   // GBK_TO_UNICODE[17068] := 16#B57B;
   // GBK_TO_UNICODE[17069] := 16#7958;
   // GBK_TO_UNICODE[17070] := 16#B57C;
   // GBK_TO_UNICODE[17071] := 16#7959;
   // GBK_TO_UNICODE[17072] := 16#B57D;
   // GBK_TO_UNICODE[17073] := 16#7961;
   // GBK_TO_UNICODE[17074] := 16#B57E;
   // GBK_TO_UNICODE[17075] := 16#7963;
   // GBK_TO_UNICODE[17076] := 16#B580;
   // GBK_TO_UNICODE[17077] := 16#7964;
   // GBK_TO_UNICODE[17078] := 16#B581;
   // GBK_TO_UNICODE[17079] := 16#7966;
   // GBK_TO_UNICODE[17080] := 16#B582;
   // GBK_TO_UNICODE[17081] := 16#7969;
   // GBK_TO_UNICODE[17082] := 16#B583;
   // GBK_TO_UNICODE[17083] := 16#796A;
   // GBK_TO_UNICODE[17084] := 16#B584;
   // GBK_TO_UNICODE[17085] := 16#796B;
   // GBK_TO_UNICODE[17086] := 16#B585;
   // GBK_TO_UNICODE[17087] := 16#796C;
   // GBK_TO_UNICODE[17088] := 16#B586;
   // GBK_TO_UNICODE[17089] := 16#796E;
   // GBK_TO_UNICODE[17090] := 16#B587;
   // GBK_TO_UNICODE[17091] := 16#7970;
   // GBK_TO_UNICODE[17092] := 16#B588;
   // GBK_TO_UNICODE[17093] := 16#7971;
   // GBK_TO_UNICODE[17094] := 16#B589;
   // GBK_TO_UNICODE[17095] := 16#7972;
   // GBK_TO_UNICODE[17096] := 16#B58A;
   // GBK_TO_UNICODE[17097] := 16#7973;
   // GBK_TO_UNICODE[17098] := 16#B58B;
   // GBK_TO_UNICODE[17099] := 16#7974;
   // GBK_TO_UNICODE[17100] := 16#B58C;
   // GBK_TO_UNICODE[17101] := 16#7975;
   // GBK_TO_UNICODE[17102] := 16#B58D;
   // GBK_TO_UNICODE[17103] := 16#7976;
   // GBK_TO_UNICODE[17104] := 16#B58E;
   // GBK_TO_UNICODE[17105] := 16#7979;
   // GBK_TO_UNICODE[17106] := 16#B58F;
   // GBK_TO_UNICODE[17107] := 16#797B;
   // GBK_TO_UNICODE[17108] := 16#B590;
   // GBK_TO_UNICODE[17109] := 16#797C;
   // GBK_TO_UNICODE[17110] := 16#B591;
   // GBK_TO_UNICODE[17111] := 16#797D;
   // GBK_TO_UNICODE[17112] := 16#B592;
   // GBK_TO_UNICODE[17113] := 16#797E;
   // GBK_TO_UNICODE[17114] := 16#B593;
   // GBK_TO_UNICODE[17115] := 16#797F;
   // GBK_TO_UNICODE[17116] := 16#B594;
   // GBK_TO_UNICODE[17117] := 16#7982;
   // GBK_TO_UNICODE[17118] := 16#B595;
   // GBK_TO_UNICODE[17119] := 16#7983;
   // GBK_TO_UNICODE[17120] := 16#B596;
   // GBK_TO_UNICODE[17121] := 16#7986;
   // GBK_TO_UNICODE[17122] := 16#B597;
   // GBK_TO_UNICODE[17123] := 16#7987;
   // GBK_TO_UNICODE[17124] := 16#B598;
   // GBK_TO_UNICODE[17125] := 16#7988;
   // GBK_TO_UNICODE[17126] := 16#B599;
   // GBK_TO_UNICODE[17127] := 16#7989;
   // GBK_TO_UNICODE[17128] := 16#B59A;
   // GBK_TO_UNICODE[17129] := 16#798B;
   // GBK_TO_UNICODE[17130] := 16#B59B;
   // GBK_TO_UNICODE[17131] := 16#798C;
   // GBK_TO_UNICODE[17132] := 16#B59C;
   // GBK_TO_UNICODE[17133] := 16#798D;
   // GBK_TO_UNICODE[17134] := 16#B59D;
   // GBK_TO_UNICODE[17135] := 16#798E;
   // GBK_TO_UNICODE[17136] := 16#B59E;
   // GBK_TO_UNICODE[17137] := 16#7990;
   // GBK_TO_UNICODE[17138] := 16#B59F;
   // GBK_TO_UNICODE[17139] := 16#7991;
   // GBK_TO_UNICODE[17140] := 16#B5A0;
   // GBK_TO_UNICODE[17141] := 16#7992;
   // GBK_TO_UNICODE[17142] := 16#B5A1;
   // GBK_TO_UNICODE[17143] := 16#6020;
   // GBK_TO_UNICODE[17144] := 16#B5A2;
   // GBK_TO_UNICODE[17145] := 16#803D;
   // GBK_TO_UNICODE[17146] := 16#B5A3;
   // GBK_TO_UNICODE[17147] := 16#62C5;
   // GBK_TO_UNICODE[17148] := 16#B5A4;
   // GBK_TO_UNICODE[17149] := 16#4E39;
   // GBK_TO_UNICODE[17150] := 16#B5A5;
   // GBK_TO_UNICODE[17151] := 16#5355;
   // GBK_TO_UNICODE[17152] := 16#B5A6;
   // GBK_TO_UNICODE[17153] := 16#90F8;
   // GBK_TO_UNICODE[17154] := 16#B5A7;
   // GBK_TO_UNICODE[17155] := 16#63B8;
   // GBK_TO_UNICODE[17156] := 16#B5A8;
   // GBK_TO_UNICODE[17157] := 16#80C6;
   // GBK_TO_UNICODE[17158] := 16#B5A9;
   // GBK_TO_UNICODE[17159] := 16#65E6;
   // GBK_TO_UNICODE[17160] := 16#B5AA;
   // GBK_TO_UNICODE[17161] := 16#6C2E;
   // GBK_TO_UNICODE[17162] := 16#B5AB;
   // GBK_TO_UNICODE[17163] := 16#4F46;
   // GBK_TO_UNICODE[17164] := 16#B5AC;
   // GBK_TO_UNICODE[17165] := 16#60EE;
   // GBK_TO_UNICODE[17166] := 16#B5AD;
   // GBK_TO_UNICODE[17167] := 16#6DE1;
   // GBK_TO_UNICODE[17168] := 16#B5AE;
   // GBK_TO_UNICODE[17169] := 16#8BDE;
   // GBK_TO_UNICODE[17170] := 16#B5AF;
   // GBK_TO_UNICODE[17171] := 16#5F39;
   // GBK_TO_UNICODE[17172] := 16#B5B0;
   // GBK_TO_UNICODE[17173] := 16#86CB;
   // GBK_TO_UNICODE[17174] := 16#B5B1;
   // GBK_TO_UNICODE[17175] := 16#5F53;
   // GBK_TO_UNICODE[17176] := 16#B5B2;
   // GBK_TO_UNICODE[17177] := 16#6321;
   // GBK_TO_UNICODE[17178] := 16#B5B3;
   // GBK_TO_UNICODE[17179] := 16#515A;
   // GBK_TO_UNICODE[17180] := 16#B5B4;
   // GBK_TO_UNICODE[17181] := 16#8361;
   // GBK_TO_UNICODE[17182] := 16#B5B5;
   // GBK_TO_UNICODE[17183] := 16#6863;
   // GBK_TO_UNICODE[17184] := 16#B5B6;
   // GBK_TO_UNICODE[17185] := 16#5200;
   // GBK_TO_UNICODE[17186] := 16#B5B7;
   // GBK_TO_UNICODE[17187] := 16#6363;
   // GBK_TO_UNICODE[17188] := 16#B5B8;
   // GBK_TO_UNICODE[17189] := 16#8E48;
   // GBK_TO_UNICODE[17190] := 16#B5B9;
   // GBK_TO_UNICODE[17191] := 16#5012;
   // GBK_TO_UNICODE[17192] := 16#B5BA;
   // GBK_TO_UNICODE[17193] := 16#5C9B;
   // GBK_TO_UNICODE[17194] := 16#B5BB;
   // GBK_TO_UNICODE[17195] := 16#7977;
   // GBK_TO_UNICODE[17196] := 16#B5BC;
   // GBK_TO_UNICODE[17197] := 16#5BFC;
   // GBK_TO_UNICODE[17198] := 16#B5BD;
   // GBK_TO_UNICODE[17199] := 16#5230;
   // GBK_TO_UNICODE[17200] := 16#B5BE;
   // GBK_TO_UNICODE[17201] := 16#7A3B;
   // GBK_TO_UNICODE[17202] := 16#B5BF;
   // GBK_TO_UNICODE[17203] := 16#60BC;
   // GBK_TO_UNICODE[17204] := 16#B5C0;
   // GBK_TO_UNICODE[17205] := 16#9053;
   // GBK_TO_UNICODE[17206] := 16#B5C1;
   // GBK_TO_UNICODE[17207] := 16#76D7;
   // GBK_TO_UNICODE[17208] := 16#B5C2;
   // GBK_TO_UNICODE[17209] := 16#5FB7;
   // GBK_TO_UNICODE[17210] := 16#B5C3;
   // GBK_TO_UNICODE[17211] := 16#5F97;
   // GBK_TO_UNICODE[17212] := 16#B5C4;
   // GBK_TO_UNICODE[17213] := 16#7684;
   // GBK_TO_UNICODE[17214] := 16#B5C5;
   // GBK_TO_UNICODE[17215] := 16#8E6C;
   // GBK_TO_UNICODE[17216] := 16#B5C6;
   // GBK_TO_UNICODE[17217] := 16#706F;
   // GBK_TO_UNICODE[17218] := 16#B5C7;
   // GBK_TO_UNICODE[17219] := 16#767B;
   // GBK_TO_UNICODE[17220] := 16#B5C8;
   // GBK_TO_UNICODE[17221] := 16#7B49;
   // GBK_TO_UNICODE[17222] := 16#B5C9;
   // GBK_TO_UNICODE[17223] := 16#77AA;
   // GBK_TO_UNICODE[17224] := 16#B5CA;
   // GBK_TO_UNICODE[17225] := 16#51F3;
   // GBK_TO_UNICODE[17226] := 16#B5CB;
   // GBK_TO_UNICODE[17227] := 16#9093;
   // GBK_TO_UNICODE[17228] := 16#B5CC;
   // GBK_TO_UNICODE[17229] := 16#5824;
   // GBK_TO_UNICODE[17230] := 16#B5CD;
   // GBK_TO_UNICODE[17231] := 16#4F4E;
   // GBK_TO_UNICODE[17232] := 16#B5CE;
   // GBK_TO_UNICODE[17233] := 16#6EF4;
   // GBK_TO_UNICODE[17234] := 16#B5CF;
   // GBK_TO_UNICODE[17235] := 16#8FEA;
   // GBK_TO_UNICODE[17236] := 16#B5D0;
   // GBK_TO_UNICODE[17237] := 16#654C;
   // GBK_TO_UNICODE[17238] := 16#B5D1;
   // GBK_TO_UNICODE[17239] := 16#7B1B;
   // GBK_TO_UNICODE[17240] := 16#B5D2;
   // GBK_TO_UNICODE[17241] := 16#72C4;
   // GBK_TO_UNICODE[17242] := 16#B5D3;
   // GBK_TO_UNICODE[17243] := 16#6DA4;
   // GBK_TO_UNICODE[17244] := 16#B5D4;
   // GBK_TO_UNICODE[17245] := 16#7FDF;
   // GBK_TO_UNICODE[17246] := 16#B5D5;
   // GBK_TO_UNICODE[17247] := 16#5AE1;
   // GBK_TO_UNICODE[17248] := 16#B5D6;
   // GBK_TO_UNICODE[17249] := 16#62B5;
   // GBK_TO_UNICODE[17250] := 16#B5D7;
   // GBK_TO_UNICODE[17251] := 16#5E95;
   // GBK_TO_UNICODE[17252] := 16#B5D8;
   // GBK_TO_UNICODE[17253] := 16#5730;
   // GBK_TO_UNICODE[17254] := 16#B5D9;
   // GBK_TO_UNICODE[17255] := 16#8482;
   // GBK_TO_UNICODE[17256] := 16#B5DA;
   // GBK_TO_UNICODE[17257] := 16#7B2C;
   // GBK_TO_UNICODE[17258] := 16#B5DB;
   // GBK_TO_UNICODE[17259] := 16#5E1D;
   // GBK_TO_UNICODE[17260] := 16#B5DC;
   // GBK_TO_UNICODE[17261] := 16#5F1F;
   // GBK_TO_UNICODE[17262] := 16#B5DD;
   // GBK_TO_UNICODE[17263] := 16#9012;
   // GBK_TO_UNICODE[17264] := 16#B5DE;
   // GBK_TO_UNICODE[17265] := 16#7F14;
   // GBK_TO_UNICODE[17266] := 16#B5DF;
   // GBK_TO_UNICODE[17267] := 16#98A0;
   // GBK_TO_UNICODE[17268] := 16#B5E0;
   // GBK_TO_UNICODE[17269] := 16#6382;
   // GBK_TO_UNICODE[17270] := 16#B5E1;
   // GBK_TO_UNICODE[17271] := 16#6EC7;
   // GBK_TO_UNICODE[17272] := 16#B5E2;
   // GBK_TO_UNICODE[17273] := 16#7898;
   // GBK_TO_UNICODE[17274] := 16#B5E3;
   // GBK_TO_UNICODE[17275] := 16#70B9;
   // GBK_TO_UNICODE[17276] := 16#B5E4;
   // GBK_TO_UNICODE[17277] := 16#5178;
   // GBK_TO_UNICODE[17278] := 16#B5E5;
   // GBK_TO_UNICODE[17279] := 16#975B;
   // GBK_TO_UNICODE[17280] := 16#B5E6;
   // GBK_TO_UNICODE[17281] := 16#57AB;
   // GBK_TO_UNICODE[17282] := 16#B5E7;
   // GBK_TO_UNICODE[17283] := 16#7535;
   // GBK_TO_UNICODE[17284] := 16#B5E8;
   // GBK_TO_UNICODE[17285] := 16#4F43;
   // GBK_TO_UNICODE[17286] := 16#B5E9;
   // GBK_TO_UNICODE[17287] := 16#7538;
   // GBK_TO_UNICODE[17288] := 16#B5EA;
   // GBK_TO_UNICODE[17289] := 16#5E97;
   // GBK_TO_UNICODE[17290] := 16#B5EB;
   // GBK_TO_UNICODE[17291] := 16#60E6;
   // GBK_TO_UNICODE[17292] := 16#B5EC;
   // GBK_TO_UNICODE[17293] := 16#5960;
   // GBK_TO_UNICODE[17294] := 16#B5ED;
   // GBK_TO_UNICODE[17295] := 16#6DC0;
   // GBK_TO_UNICODE[17296] := 16#B5EE;
   // GBK_TO_UNICODE[17297] := 16#6BBF;
   // GBK_TO_UNICODE[17298] := 16#B5EF;
   // GBK_TO_UNICODE[17299] := 16#7889;
   // GBK_TO_UNICODE[17300] := 16#B5F0;
   // GBK_TO_UNICODE[17301] := 16#53FC;
   // GBK_TO_UNICODE[17302] := 16#B5F1;
   // GBK_TO_UNICODE[17303] := 16#96D5;
   // GBK_TO_UNICODE[17304] := 16#B5F2;
   // GBK_TO_UNICODE[17305] := 16#51CB;
   // GBK_TO_UNICODE[17306] := 16#B5F3;
   // GBK_TO_UNICODE[17307] := 16#5201;
   // GBK_TO_UNICODE[17308] := 16#B5F4;
   // GBK_TO_UNICODE[17309] := 16#6389;
   // GBK_TO_UNICODE[17310] := 16#B5F5;
   // GBK_TO_UNICODE[17311] := 16#540A;
   // GBK_TO_UNICODE[17312] := 16#B5F6;
   // GBK_TO_UNICODE[17313] := 16#9493;
   // GBK_TO_UNICODE[17314] := 16#B5F7;
   // GBK_TO_UNICODE[17315] := 16#8C03;
   // GBK_TO_UNICODE[17316] := 16#B5F8;
   // GBK_TO_UNICODE[17317] := 16#8DCC;
   // GBK_TO_UNICODE[17318] := 16#B5F9;
   // GBK_TO_UNICODE[17319] := 16#7239;
   // GBK_TO_UNICODE[17320] := 16#B5FA;
   // GBK_TO_UNICODE[17321] := 16#789F;
   // GBK_TO_UNICODE[17322] := 16#B5FB;
   // GBK_TO_UNICODE[17323] := 16#8776;
   // GBK_TO_UNICODE[17324] := 16#B5FC;
   // GBK_TO_UNICODE[17325] := 16#8FED;
   // GBK_TO_UNICODE[17326] := 16#B5FD;
   // GBK_TO_UNICODE[17327] := 16#8C0D;
   // GBK_TO_UNICODE[17328] := 16#B5FE;
   // GBK_TO_UNICODE[17329] := 16#53E0;
   // GBK_TO_UNICODE[17330] := 16#B640;
   // GBK_TO_UNICODE[17331] := 16#7993;
   // GBK_TO_UNICODE[17332] := 16#B641;
   // GBK_TO_UNICODE[17333] := 16#7994;
   // GBK_TO_UNICODE[17334] := 16#B642;
   // GBK_TO_UNICODE[17335] := 16#7995;
   // GBK_TO_UNICODE[17336] := 16#B643;
   // GBK_TO_UNICODE[17337] := 16#7996;
   // GBK_TO_UNICODE[17338] := 16#B644;
   // GBK_TO_UNICODE[17339] := 16#7997;
   // GBK_TO_UNICODE[17340] := 16#B645;
   // GBK_TO_UNICODE[17341] := 16#7998;
   // GBK_TO_UNICODE[17342] := 16#B646;
   // GBK_TO_UNICODE[17343] := 16#7999;
   // GBK_TO_UNICODE[17344] := 16#B647;
   // GBK_TO_UNICODE[17345] := 16#799B;
   // GBK_TO_UNICODE[17346] := 16#B648;
   // GBK_TO_UNICODE[17347] := 16#799C;
   // GBK_TO_UNICODE[17348] := 16#B649;
   // GBK_TO_UNICODE[17349] := 16#799D;
   // GBK_TO_UNICODE[17350] := 16#B64A;
   // GBK_TO_UNICODE[17351] := 16#799E;
   // GBK_TO_UNICODE[17352] := 16#B64B;
   // GBK_TO_UNICODE[17353] := 16#799F;
   // GBK_TO_UNICODE[17354] := 16#B64C;
   // GBK_TO_UNICODE[17355] := 16#79A0;
   // GBK_TO_UNICODE[17356] := 16#B64D;
   // GBK_TO_UNICODE[17357] := 16#79A1;
   // GBK_TO_UNICODE[17358] := 16#B64E;
   // GBK_TO_UNICODE[17359] := 16#79A2;
   // GBK_TO_UNICODE[17360] := 16#B64F;
   // GBK_TO_UNICODE[17361] := 16#79A3;
   // GBK_TO_UNICODE[17362] := 16#B650;
   // GBK_TO_UNICODE[17363] := 16#79A4;
   // GBK_TO_UNICODE[17364] := 16#B651;
   // GBK_TO_UNICODE[17365] := 16#79A5;
   // GBK_TO_UNICODE[17366] := 16#B652;
   // GBK_TO_UNICODE[17367] := 16#79A6;
   // GBK_TO_UNICODE[17368] := 16#B653;
   // GBK_TO_UNICODE[17369] := 16#79A8;
   // GBK_TO_UNICODE[17370] := 16#B654;
   // GBK_TO_UNICODE[17371] := 16#79A9;
   // GBK_TO_UNICODE[17372] := 16#B655;
   // GBK_TO_UNICODE[17373] := 16#79AA;
   // GBK_TO_UNICODE[17374] := 16#B656;
   // GBK_TO_UNICODE[17375] := 16#79AB;
   // GBK_TO_UNICODE[17376] := 16#B657;
   // GBK_TO_UNICODE[17377] := 16#79AC;
   // GBK_TO_UNICODE[17378] := 16#B658;
   // GBK_TO_UNICODE[17379] := 16#79AD;
   // GBK_TO_UNICODE[17380] := 16#B659;
   // GBK_TO_UNICODE[17381] := 16#79AE;
   // GBK_TO_UNICODE[17382] := 16#B65A;
   // GBK_TO_UNICODE[17383] := 16#79AF;
   // GBK_TO_UNICODE[17384] := 16#B65B;
   // GBK_TO_UNICODE[17385] := 16#79B0;
   // GBK_TO_UNICODE[17386] := 16#B65C;
   // GBK_TO_UNICODE[17387] := 16#79B1;
   // GBK_TO_UNICODE[17388] := 16#B65D;
   // GBK_TO_UNICODE[17389] := 16#79B2;
   // GBK_TO_UNICODE[17390] := 16#B65E;
   // GBK_TO_UNICODE[17391] := 16#79B4;
   // GBK_TO_UNICODE[17392] := 16#B65F;
   // GBK_TO_UNICODE[17393] := 16#79B5;
   // GBK_TO_UNICODE[17394] := 16#B660;
   // GBK_TO_UNICODE[17395] := 16#79B6;
   // GBK_TO_UNICODE[17396] := 16#B661;
   // GBK_TO_UNICODE[17397] := 16#79B7;
   // GBK_TO_UNICODE[17398] := 16#B662;
   // GBK_TO_UNICODE[17399] := 16#79B8;
   // GBK_TO_UNICODE[17400] := 16#B663;
   // GBK_TO_UNICODE[17401] := 16#79BC;
   // GBK_TO_UNICODE[17402] := 16#B664;
   // GBK_TO_UNICODE[17403] := 16#79BF;
   // GBK_TO_UNICODE[17404] := 16#B665;
   // GBK_TO_UNICODE[17405] := 16#79C2;
   // GBK_TO_UNICODE[17406] := 16#B666;
   // GBK_TO_UNICODE[17407] := 16#79C4;
   // GBK_TO_UNICODE[17408] := 16#B667;
   // GBK_TO_UNICODE[17409] := 16#79C5;
   // GBK_TO_UNICODE[17410] := 16#B668;
   // GBK_TO_UNICODE[17411] := 16#79C7;
   // GBK_TO_UNICODE[17412] := 16#B669;
   // GBK_TO_UNICODE[17413] := 16#79C8;
   // GBK_TO_UNICODE[17414] := 16#B66A;
   // GBK_TO_UNICODE[17415] := 16#79CA;
   // GBK_TO_UNICODE[17416] := 16#B66B;
   // GBK_TO_UNICODE[17417] := 16#79CC;
   // GBK_TO_UNICODE[17418] := 16#B66C;
   // GBK_TO_UNICODE[17419] := 16#79CE;
   // GBK_TO_UNICODE[17420] := 16#B66D;
   // GBK_TO_UNICODE[17421] := 16#79CF;
   // GBK_TO_UNICODE[17422] := 16#B66E;
   // GBK_TO_UNICODE[17423] := 16#79D0;
   // GBK_TO_UNICODE[17424] := 16#B66F;
   // GBK_TO_UNICODE[17425] := 16#79D3;
   // GBK_TO_UNICODE[17426] := 16#B670;
   // GBK_TO_UNICODE[17427] := 16#79D4;
   // GBK_TO_UNICODE[17428] := 16#B671;
   // GBK_TO_UNICODE[17429] := 16#79D6;
   // GBK_TO_UNICODE[17430] := 16#B672;
   // GBK_TO_UNICODE[17431] := 16#79D7;
   // GBK_TO_UNICODE[17432] := 16#B673;
   // GBK_TO_UNICODE[17433] := 16#79D9;
   // GBK_TO_UNICODE[17434] := 16#B674;
   // GBK_TO_UNICODE[17435] := 16#79DA;
   // GBK_TO_UNICODE[17436] := 16#B675;
   // GBK_TO_UNICODE[17437] := 16#79DB;
   // GBK_TO_UNICODE[17438] := 16#B676;
   // GBK_TO_UNICODE[17439] := 16#79DC;
   // GBK_TO_UNICODE[17440] := 16#B677;
   // GBK_TO_UNICODE[17441] := 16#79DD;
   // GBK_TO_UNICODE[17442] := 16#B678;
   // GBK_TO_UNICODE[17443] := 16#79DE;
   // GBK_TO_UNICODE[17444] := 16#B679;
   // GBK_TO_UNICODE[17445] := 16#79E0;
   // GBK_TO_UNICODE[17446] := 16#B67A;
   // GBK_TO_UNICODE[17447] := 16#79E1;
   // GBK_TO_UNICODE[17448] := 16#B67B;
   // GBK_TO_UNICODE[17449] := 16#79E2;
   // GBK_TO_UNICODE[17450] := 16#B67C;
   // GBK_TO_UNICODE[17451] := 16#79E5;
   // GBK_TO_UNICODE[17452] := 16#B67D;
   // GBK_TO_UNICODE[17453] := 16#79E8;
   // GBK_TO_UNICODE[17454] := 16#B67E;
   // GBK_TO_UNICODE[17455] := 16#79EA;
   // GBK_TO_UNICODE[17456] := 16#B680;
   // GBK_TO_UNICODE[17457] := 16#79EC;
   // GBK_TO_UNICODE[17458] := 16#B681;
   // GBK_TO_UNICODE[17459] := 16#79EE;
   // GBK_TO_UNICODE[17460] := 16#B682;
   // GBK_TO_UNICODE[17461] := 16#79F1;
   // GBK_TO_UNICODE[17462] := 16#B683;
   // GBK_TO_UNICODE[17463] := 16#79F2;
   // GBK_TO_UNICODE[17464] := 16#B684;
   // GBK_TO_UNICODE[17465] := 16#79F3;
   // GBK_TO_UNICODE[17466] := 16#B685;
   // GBK_TO_UNICODE[17467] := 16#79F4;
   // GBK_TO_UNICODE[17468] := 16#B686;
   // GBK_TO_UNICODE[17469] := 16#79F5;
   // GBK_TO_UNICODE[17470] := 16#B687;
   // GBK_TO_UNICODE[17471] := 16#79F6;
   // GBK_TO_UNICODE[17472] := 16#B688;
   // GBK_TO_UNICODE[17473] := 16#79F7;
   // GBK_TO_UNICODE[17474] := 16#B689;
   // GBK_TO_UNICODE[17475] := 16#79F9;
   // GBK_TO_UNICODE[17476] := 16#B68A;
   // GBK_TO_UNICODE[17477] := 16#79FA;
   // GBK_TO_UNICODE[17478] := 16#B68B;
   // GBK_TO_UNICODE[17479] := 16#79FC;
   // GBK_TO_UNICODE[17480] := 16#B68C;
   // GBK_TO_UNICODE[17481] := 16#79FE;
   // GBK_TO_UNICODE[17482] := 16#B68D;
   // GBK_TO_UNICODE[17483] := 16#79FF;
   // GBK_TO_UNICODE[17484] := 16#B68E;
   // GBK_TO_UNICODE[17485] := 16#7A01;
   // GBK_TO_UNICODE[17486] := 16#B68F;
   // GBK_TO_UNICODE[17487] := 16#7A04;
   // GBK_TO_UNICODE[17488] := 16#B690;
   // GBK_TO_UNICODE[17489] := 16#7A05;
   // GBK_TO_UNICODE[17490] := 16#B691;
   // GBK_TO_UNICODE[17491] := 16#7A07;
   // GBK_TO_UNICODE[17492] := 16#B692;
   // GBK_TO_UNICODE[17493] := 16#7A08;
   // GBK_TO_UNICODE[17494] := 16#B693;
   // GBK_TO_UNICODE[17495] := 16#7A09;
   // GBK_TO_UNICODE[17496] := 16#B694;
   // GBK_TO_UNICODE[17497] := 16#7A0A;
   // GBK_TO_UNICODE[17498] := 16#B695;
   // GBK_TO_UNICODE[17499] := 16#7A0C;
   // GBK_TO_UNICODE[17500] := 16#B696;
   // GBK_TO_UNICODE[17501] := 16#7A0F;
   // GBK_TO_UNICODE[17502] := 16#B697;
   // GBK_TO_UNICODE[17503] := 16#7A10;
   // GBK_TO_UNICODE[17504] := 16#B698;
   // GBK_TO_UNICODE[17505] := 16#7A11;
   // GBK_TO_UNICODE[17506] := 16#B699;
   // GBK_TO_UNICODE[17507] := 16#7A12;
   // GBK_TO_UNICODE[17508] := 16#B69A;
   // GBK_TO_UNICODE[17509] := 16#7A13;
   // GBK_TO_UNICODE[17510] := 16#B69B;
   // GBK_TO_UNICODE[17511] := 16#7A15;
   // GBK_TO_UNICODE[17512] := 16#B69C;
   // GBK_TO_UNICODE[17513] := 16#7A16;
   // GBK_TO_UNICODE[17514] := 16#B69D;
   // GBK_TO_UNICODE[17515] := 16#7A18;
   // GBK_TO_UNICODE[17516] := 16#B69E;
   // GBK_TO_UNICODE[17517] := 16#7A19;
   // GBK_TO_UNICODE[17518] := 16#B69F;
   // GBK_TO_UNICODE[17519] := 16#7A1B;
   // GBK_TO_UNICODE[17520] := 16#B6A0;
   // GBK_TO_UNICODE[17521] := 16#7A1C;
   // GBK_TO_UNICODE[17522] := 16#B6A1;
   // GBK_TO_UNICODE[17523] := 16#4E01;
   // GBK_TO_UNICODE[17524] := 16#B6A2;
   // GBK_TO_UNICODE[17525] := 16#76EF;
   // GBK_TO_UNICODE[17526] := 16#B6A3;
   // GBK_TO_UNICODE[17527] := 16#53EE;
   // GBK_TO_UNICODE[17528] := 16#B6A4;
   // GBK_TO_UNICODE[17529] := 16#9489;
   // GBK_TO_UNICODE[17530] := 16#B6A5;
   // GBK_TO_UNICODE[17531] := 16#9876;
   // GBK_TO_UNICODE[17532] := 16#B6A6;
   // GBK_TO_UNICODE[17533] := 16#9F0E;
   // GBK_TO_UNICODE[17534] := 16#B6A7;
   // GBK_TO_UNICODE[17535] := 16#952D;
   // GBK_TO_UNICODE[17536] := 16#B6A8;
   // GBK_TO_UNICODE[17537] := 16#5B9A;
   // GBK_TO_UNICODE[17538] := 16#B6A9;
   // GBK_TO_UNICODE[17539] := 16#8BA2;
   // GBK_TO_UNICODE[17540] := 16#B6AA;
   // GBK_TO_UNICODE[17541] := 16#4E22;
   // GBK_TO_UNICODE[17542] := 16#B6AB;
   // GBK_TO_UNICODE[17543] := 16#4E1C;
   // GBK_TO_UNICODE[17544] := 16#B6AC;
   // GBK_TO_UNICODE[17545] := 16#51AC;
   // GBK_TO_UNICODE[17546] := 16#B6AD;
   // GBK_TO_UNICODE[17547] := 16#8463;
   // GBK_TO_UNICODE[17548] := 16#B6AE;
   // GBK_TO_UNICODE[17549] := 16#61C2;
   // GBK_TO_UNICODE[17550] := 16#B6AF;
   // GBK_TO_UNICODE[17551] := 16#52A8;
   // GBK_TO_UNICODE[17552] := 16#B6B0;
   // GBK_TO_UNICODE[17553] := 16#680B;
   // GBK_TO_UNICODE[17554] := 16#B6B1;
   // GBK_TO_UNICODE[17555] := 16#4F97;
   // GBK_TO_UNICODE[17556] := 16#B6B2;
   // GBK_TO_UNICODE[17557] := 16#606B;
   // GBK_TO_UNICODE[17558] := 16#B6B3;
   // GBK_TO_UNICODE[17559] := 16#51BB;
   // GBK_TO_UNICODE[17560] := 16#B6B4;
   // GBK_TO_UNICODE[17561] := 16#6D1E;
   // GBK_TO_UNICODE[17562] := 16#B6B5;
   // GBK_TO_UNICODE[17563] := 16#515C;
   // GBK_TO_UNICODE[17564] := 16#B6B6;
   // GBK_TO_UNICODE[17565] := 16#6296;
   // GBK_TO_UNICODE[17566] := 16#B6B7;
   // GBK_TO_UNICODE[17567] := 16#6597;
   // GBK_TO_UNICODE[17568] := 16#B6B8;
   // GBK_TO_UNICODE[17569] := 16#9661;
   // GBK_TO_UNICODE[17570] := 16#B6B9;
   // GBK_TO_UNICODE[17571] := 16#8C46;
   // GBK_TO_UNICODE[17572] := 16#B6BA;
   // GBK_TO_UNICODE[17573] := 16#9017;
   // GBK_TO_UNICODE[17574] := 16#B6BB;
   // GBK_TO_UNICODE[17575] := 16#75D8;
   // GBK_TO_UNICODE[17576] := 16#B6BC;
   // GBK_TO_UNICODE[17577] := 16#90FD;
   // GBK_TO_UNICODE[17578] := 16#B6BD;
   // GBK_TO_UNICODE[17579] := 16#7763;
   // GBK_TO_UNICODE[17580] := 16#B6BE;
   // GBK_TO_UNICODE[17581] := 16#6BD2;
   // GBK_TO_UNICODE[17582] := 16#B6BF;
   // GBK_TO_UNICODE[17583] := 16#728A;
   // GBK_TO_UNICODE[17584] := 16#B6C0;
   // GBK_TO_UNICODE[17585] := 16#72EC;
   // GBK_TO_UNICODE[17586] := 16#B6C1;
   // GBK_TO_UNICODE[17587] := 16#8BFB;
   // GBK_TO_UNICODE[17588] := 16#B6C2;
   // GBK_TO_UNICODE[17589] := 16#5835;
   // GBK_TO_UNICODE[17590] := 16#B6C3;
   // GBK_TO_UNICODE[17591] := 16#7779;
   // GBK_TO_UNICODE[17592] := 16#B6C4;
   // GBK_TO_UNICODE[17593] := 16#8D4C;
   // GBK_TO_UNICODE[17594] := 16#B6C5;
   // GBK_TO_UNICODE[17595] := 16#675C;
   // GBK_TO_UNICODE[17596] := 16#B6C6;
   // GBK_TO_UNICODE[17597] := 16#9540;
   // GBK_TO_UNICODE[17598] := 16#B6C7;
   // GBK_TO_UNICODE[17599] := 16#809A;
   // GBK_TO_UNICODE[17600] := 16#B6C8;
   // GBK_TO_UNICODE[17601] := 16#5EA6;
   // GBK_TO_UNICODE[17602] := 16#B6C9;
   // GBK_TO_UNICODE[17603] := 16#6E21;
   // GBK_TO_UNICODE[17604] := 16#B6CA;
   // GBK_TO_UNICODE[17605] := 16#5992;
   // GBK_TO_UNICODE[17606] := 16#B6CB;
   // GBK_TO_UNICODE[17607] := 16#7AEF;
   // GBK_TO_UNICODE[17608] := 16#B6CC;
   // GBK_TO_UNICODE[17609] := 16#77ED;
   // GBK_TO_UNICODE[17610] := 16#B6CD;
   // GBK_TO_UNICODE[17611] := 16#953B;
   // GBK_TO_UNICODE[17612] := 16#B6CE;
   // GBK_TO_UNICODE[17613] := 16#6BB5;
   // GBK_TO_UNICODE[17614] := 16#B6CF;
   // GBK_TO_UNICODE[17615] := 16#65AD;
   // GBK_TO_UNICODE[17616] := 16#B6D0;
   // GBK_TO_UNICODE[17617] := 16#7F0E;
   // GBK_TO_UNICODE[17618] := 16#B6D1;
   // GBK_TO_UNICODE[17619] := 16#5806;
   // GBK_TO_UNICODE[17620] := 16#B6D2;
   // GBK_TO_UNICODE[17621] := 16#5151;
   // GBK_TO_UNICODE[17622] := 16#B6D3;
   // GBK_TO_UNICODE[17623] := 16#961F;
   // GBK_TO_UNICODE[17624] := 16#B6D4;
   // GBK_TO_UNICODE[17625] := 16#5BF9;
   // GBK_TO_UNICODE[17626] := 16#B6D5;
   // GBK_TO_UNICODE[17627] := 16#58A9;
   // GBK_TO_UNICODE[17628] := 16#B6D6;
   // GBK_TO_UNICODE[17629] := 16#5428;
   // GBK_TO_UNICODE[17630] := 16#B6D7;
   // GBK_TO_UNICODE[17631] := 16#8E72;
   // GBK_TO_UNICODE[17632] := 16#B6D8;
   // GBK_TO_UNICODE[17633] := 16#6566;
   // GBK_TO_UNICODE[17634] := 16#B6D9;
   // GBK_TO_UNICODE[17635] := 16#987F;
   // GBK_TO_UNICODE[17636] := 16#B6DA;
   // GBK_TO_UNICODE[17637] := 16#56E4;
   // GBK_TO_UNICODE[17638] := 16#B6DB;
   // GBK_TO_UNICODE[17639] := 16#949D;
   // GBK_TO_UNICODE[17640] := 16#B6DC;
   // GBK_TO_UNICODE[17641] := 16#76FE;
   // GBK_TO_UNICODE[17642] := 16#B6DD;
   // GBK_TO_UNICODE[17643] := 16#9041;
   // GBK_TO_UNICODE[17644] := 16#B6DE;
   // GBK_TO_UNICODE[17645] := 16#6387;
   // GBK_TO_UNICODE[17646] := 16#B6DF;
   // GBK_TO_UNICODE[17647] := 16#54C6;
   // GBK_TO_UNICODE[17648] := 16#B6E0;
   // GBK_TO_UNICODE[17649] := 16#591A;
   // GBK_TO_UNICODE[17650] := 16#B6E1;
   // GBK_TO_UNICODE[17651] := 16#593A;
   // GBK_TO_UNICODE[17652] := 16#B6E2;
   // GBK_TO_UNICODE[17653] := 16#579B;
   // GBK_TO_UNICODE[17654] := 16#B6E3;
   // GBK_TO_UNICODE[17655] := 16#8EB2;
   // GBK_TO_UNICODE[17656] := 16#B6E4;
   // GBK_TO_UNICODE[17657] := 16#6735;
   // GBK_TO_UNICODE[17658] := 16#B6E5;
   // GBK_TO_UNICODE[17659] := 16#8DFA;
   // GBK_TO_UNICODE[17660] := 16#B6E6;
   // GBK_TO_UNICODE[17661] := 16#8235;
   // GBK_TO_UNICODE[17662] := 16#B6E7;
   // GBK_TO_UNICODE[17663] := 16#5241;
   // GBK_TO_UNICODE[17664] := 16#B6E8;
   // GBK_TO_UNICODE[17665] := 16#60F0;
   // GBK_TO_UNICODE[17666] := 16#B6E9;
   // GBK_TO_UNICODE[17667] := 16#5815;
   // GBK_TO_UNICODE[17668] := 16#B6EA;
   // GBK_TO_UNICODE[17669] := 16#86FE;
   // GBK_TO_UNICODE[17670] := 16#B6EB;
   // GBK_TO_UNICODE[17671] := 16#5CE8;
   // GBK_TO_UNICODE[17672] := 16#B6EC;
   // GBK_TO_UNICODE[17673] := 16#9E45;
   // GBK_TO_UNICODE[17674] := 16#B6ED;
   // GBK_TO_UNICODE[17675] := 16#4FC4;
   // GBK_TO_UNICODE[17676] := 16#B6EE;
   // GBK_TO_UNICODE[17677] := 16#989D;
   // GBK_TO_UNICODE[17678] := 16#B6EF;
   // GBK_TO_UNICODE[17679] := 16#8BB9;
   // GBK_TO_UNICODE[17680] := 16#B6F0;
   // GBK_TO_UNICODE[17681] := 16#5A25;
   // GBK_TO_UNICODE[17682] := 16#B6F1;
   // GBK_TO_UNICODE[17683] := 16#6076;
   // GBK_TO_UNICODE[17684] := 16#B6F2;
   // GBK_TO_UNICODE[17685] := 16#5384;
   // GBK_TO_UNICODE[17686] := 16#B6F3;
   // GBK_TO_UNICODE[17687] := 16#627C;
   // GBK_TO_UNICODE[17688] := 16#B6F4;
   // GBK_TO_UNICODE[17689] := 16#904F;
   // GBK_TO_UNICODE[17690] := 16#B6F5;
   // GBK_TO_UNICODE[17691] := 16#9102;
   // GBK_TO_UNICODE[17692] := 16#B6F6;
   // GBK_TO_UNICODE[17693] := 16#997F;
   // GBK_TO_UNICODE[17694] := 16#B6F7;
   // GBK_TO_UNICODE[17695] := 16#6069;
   // GBK_TO_UNICODE[17696] := 16#B6F8;
   // GBK_TO_UNICODE[17697] := 16#800C;
   // GBK_TO_UNICODE[17698] := 16#B6F9;
   // GBK_TO_UNICODE[17699] := 16#513F;
   // GBK_TO_UNICODE[17700] := 16#B6FA;
   // GBK_TO_UNICODE[17701] := 16#8033;
   // GBK_TO_UNICODE[17702] := 16#B6FB;
   // GBK_TO_UNICODE[17703] := 16#5C14;
   // GBK_TO_UNICODE[17704] := 16#B6FC;
   // GBK_TO_UNICODE[17705] := 16#9975;
   // GBK_TO_UNICODE[17706] := 16#B6FD;
   // GBK_TO_UNICODE[17707] := 16#6D31;
   // GBK_TO_UNICODE[17708] := 16#B6FE;
   // GBK_TO_UNICODE[17709] := 16#4E8C;
   // GBK_TO_UNICODE[17710] := 16#B740;
   // GBK_TO_UNICODE[17711] := 16#7A1D;
   // GBK_TO_UNICODE[17712] := 16#B741;
   // GBK_TO_UNICODE[17713] := 16#7A1F;
   // GBK_TO_UNICODE[17714] := 16#B742;
   // GBK_TO_UNICODE[17715] := 16#7A21;
   // GBK_TO_UNICODE[17716] := 16#B743;
   // GBK_TO_UNICODE[17717] := 16#7A22;
   // GBK_TO_UNICODE[17718] := 16#B744;
   // GBK_TO_UNICODE[17719] := 16#7A24;
   // GBK_TO_UNICODE[17720] := 16#B745;
   // GBK_TO_UNICODE[17721] := 16#7A25;
   // GBK_TO_UNICODE[17722] := 16#B746;
   // GBK_TO_UNICODE[17723] := 16#7A26;
   // GBK_TO_UNICODE[17724] := 16#B747;
   // GBK_TO_UNICODE[17725] := 16#7A27;
   // GBK_TO_UNICODE[17726] := 16#B748;
   // GBK_TO_UNICODE[17727] := 16#7A28;
   // GBK_TO_UNICODE[17728] := 16#B749;
   // GBK_TO_UNICODE[17729] := 16#7A29;
   // GBK_TO_UNICODE[17730] := 16#B74A;
   // GBK_TO_UNICODE[17731] := 16#7A2A;
   // GBK_TO_UNICODE[17732] := 16#B74B;
   // GBK_TO_UNICODE[17733] := 16#7A2B;
   // GBK_TO_UNICODE[17734] := 16#B74C;
   // GBK_TO_UNICODE[17735] := 16#7A2C;
   // GBK_TO_UNICODE[17736] := 16#B74D;
   // GBK_TO_UNICODE[17737] := 16#7A2D;
   // GBK_TO_UNICODE[17738] := 16#B74E;
   // GBK_TO_UNICODE[17739] := 16#7A2E;
   // GBK_TO_UNICODE[17740] := 16#B74F;
   // GBK_TO_UNICODE[17741] := 16#7A2F;
   // GBK_TO_UNICODE[17742] := 16#B750;
   // GBK_TO_UNICODE[17743] := 16#7A30;
   // GBK_TO_UNICODE[17744] := 16#B751;
   // GBK_TO_UNICODE[17745] := 16#7A31;
   // GBK_TO_UNICODE[17746] := 16#B752;
   // GBK_TO_UNICODE[17747] := 16#7A32;
   // GBK_TO_UNICODE[17748] := 16#B753;
   // GBK_TO_UNICODE[17749] := 16#7A34;
   // GBK_TO_UNICODE[17750] := 16#B754;
   // GBK_TO_UNICODE[17751] := 16#7A35;
   // GBK_TO_UNICODE[17752] := 16#B755;
   // GBK_TO_UNICODE[17753] := 16#7A36;
   // GBK_TO_UNICODE[17754] := 16#B756;
   // GBK_TO_UNICODE[17755] := 16#7A38;
   // GBK_TO_UNICODE[17756] := 16#B757;
   // GBK_TO_UNICODE[17757] := 16#7A3A;
   // GBK_TO_UNICODE[17758] := 16#B758;
   // GBK_TO_UNICODE[17759] := 16#7A3E;
   // GBK_TO_UNICODE[17760] := 16#B759;
   // GBK_TO_UNICODE[17761] := 16#7A40;
   // GBK_TO_UNICODE[17762] := 16#B75A;
   // GBK_TO_UNICODE[17763] := 16#7A41;
   // GBK_TO_UNICODE[17764] := 16#B75B;
   // GBK_TO_UNICODE[17765] := 16#7A42;
   // GBK_TO_UNICODE[17766] := 16#B75C;
   // GBK_TO_UNICODE[17767] := 16#7A43;
   // GBK_TO_UNICODE[17768] := 16#B75D;
   // GBK_TO_UNICODE[17769] := 16#7A44;
   // GBK_TO_UNICODE[17770] := 16#B75E;
   // GBK_TO_UNICODE[17771] := 16#7A45;
   // GBK_TO_UNICODE[17772] := 16#B75F;
   // GBK_TO_UNICODE[17773] := 16#7A47;
   // GBK_TO_UNICODE[17774] := 16#B760;
   // GBK_TO_UNICODE[17775] := 16#7A48;
   // GBK_TO_UNICODE[17776] := 16#B761;
   // GBK_TO_UNICODE[17777] := 16#7A49;
   // GBK_TO_UNICODE[17778] := 16#B762;
   // GBK_TO_UNICODE[17779] := 16#7A4A;
   // GBK_TO_UNICODE[17780] := 16#B763;
   // GBK_TO_UNICODE[17781] := 16#7A4B;
   // GBK_TO_UNICODE[17782] := 16#B764;
   // GBK_TO_UNICODE[17783] := 16#7A4C;
   // GBK_TO_UNICODE[17784] := 16#B765;
   // GBK_TO_UNICODE[17785] := 16#7A4D;
   // GBK_TO_UNICODE[17786] := 16#B766;
   // GBK_TO_UNICODE[17787] := 16#7A4E;
   // GBK_TO_UNICODE[17788] := 16#B767;
   // GBK_TO_UNICODE[17789] := 16#7A4F;
   // GBK_TO_UNICODE[17790] := 16#B768;
   // GBK_TO_UNICODE[17791] := 16#7A50;
   // GBK_TO_UNICODE[17792] := 16#B769;
   // GBK_TO_UNICODE[17793] := 16#7A52;
   // GBK_TO_UNICODE[17794] := 16#B76A;
   // GBK_TO_UNICODE[17795] := 16#7A53;
   // GBK_TO_UNICODE[17796] := 16#B76B;
   // GBK_TO_UNICODE[17797] := 16#7A54;
   // GBK_TO_UNICODE[17798] := 16#B76C;
   // GBK_TO_UNICODE[17799] := 16#7A55;
   // GBK_TO_UNICODE[17800] := 16#B76D;
   // GBK_TO_UNICODE[17801] := 16#7A56;
   // GBK_TO_UNICODE[17802] := 16#B76E;
   // GBK_TO_UNICODE[17803] := 16#7A58;
   // GBK_TO_UNICODE[17804] := 16#B76F;
   // GBK_TO_UNICODE[17805] := 16#7A59;
   // GBK_TO_UNICODE[17806] := 16#B770;
   // GBK_TO_UNICODE[17807] := 16#7A5A;
   // GBK_TO_UNICODE[17808] := 16#B771;
   // GBK_TO_UNICODE[17809] := 16#7A5B;
   // GBK_TO_UNICODE[17810] := 16#B772;
   // GBK_TO_UNICODE[17811] := 16#7A5C;
   // GBK_TO_UNICODE[17812] := 16#B773;
   // GBK_TO_UNICODE[17813] := 16#7A5D;
   // GBK_TO_UNICODE[17814] := 16#B774;
   // GBK_TO_UNICODE[17815] := 16#7A5E;
   // GBK_TO_UNICODE[17816] := 16#B775;
   // GBK_TO_UNICODE[17817] := 16#7A5F;
   // GBK_TO_UNICODE[17818] := 16#B776;
   // GBK_TO_UNICODE[17819] := 16#7A60;
   // GBK_TO_UNICODE[17820] := 16#B777;
   // GBK_TO_UNICODE[17821] := 16#7A61;
   // GBK_TO_UNICODE[17822] := 16#B778;
   // GBK_TO_UNICODE[17823] := 16#7A62;
   // GBK_TO_UNICODE[17824] := 16#B779;
   // GBK_TO_UNICODE[17825] := 16#7A63;
   // GBK_TO_UNICODE[17826] := 16#B77A;
   // GBK_TO_UNICODE[17827] := 16#7A64;
   // GBK_TO_UNICODE[17828] := 16#B77B;
   // GBK_TO_UNICODE[17829] := 16#7A65;
   // GBK_TO_UNICODE[17830] := 16#B77C;
   // GBK_TO_UNICODE[17831] := 16#7A66;
   // GBK_TO_UNICODE[17832] := 16#B77D;
   // GBK_TO_UNICODE[17833] := 16#7A67;
   // GBK_TO_UNICODE[17834] := 16#B77E;
   // GBK_TO_UNICODE[17835] := 16#7A68;
   // GBK_TO_UNICODE[17836] := 16#B780;
   // GBK_TO_UNICODE[17837] := 16#7A69;
   // GBK_TO_UNICODE[17838] := 16#B781;
   // GBK_TO_UNICODE[17839] := 16#7A6A;
   // GBK_TO_UNICODE[17840] := 16#B782;
   // GBK_TO_UNICODE[17841] := 16#7A6B;
   // GBK_TO_UNICODE[17842] := 16#B783;
   // GBK_TO_UNICODE[17843] := 16#7A6C;
   // GBK_TO_UNICODE[17844] := 16#B784;
   // GBK_TO_UNICODE[17845] := 16#7A6D;
   // GBK_TO_UNICODE[17846] := 16#B785;
   // GBK_TO_UNICODE[17847] := 16#7A6E;
   // GBK_TO_UNICODE[17848] := 16#B786;
   // GBK_TO_UNICODE[17849] := 16#7A6F;
   // GBK_TO_UNICODE[17850] := 16#B787;
   // GBK_TO_UNICODE[17851] := 16#7A71;
   // GBK_TO_UNICODE[17852] := 16#B788;
   // GBK_TO_UNICODE[17853] := 16#7A72;
   // GBK_TO_UNICODE[17854] := 16#B789;
   // GBK_TO_UNICODE[17855] := 16#7A73;
   // GBK_TO_UNICODE[17856] := 16#B78A;
   // GBK_TO_UNICODE[17857] := 16#7A75;
   // GBK_TO_UNICODE[17858] := 16#B78B;
   // GBK_TO_UNICODE[17859] := 16#7A7B;
   // GBK_TO_UNICODE[17860] := 16#B78C;
   // GBK_TO_UNICODE[17861] := 16#7A7C;
   // GBK_TO_UNICODE[17862] := 16#B78D;
   // GBK_TO_UNICODE[17863] := 16#7A7D;
   // GBK_TO_UNICODE[17864] := 16#B78E;
   // GBK_TO_UNICODE[17865] := 16#7A7E;
   // GBK_TO_UNICODE[17866] := 16#B78F;
   // GBK_TO_UNICODE[17867] := 16#7A82;
   // GBK_TO_UNICODE[17868] := 16#B790;
   // GBK_TO_UNICODE[17869] := 16#7A85;
   // GBK_TO_UNICODE[17870] := 16#B791;
   // GBK_TO_UNICODE[17871] := 16#7A87;
   // GBK_TO_UNICODE[17872] := 16#B792;
   // GBK_TO_UNICODE[17873] := 16#7A89;
   // GBK_TO_UNICODE[17874] := 16#B793;
   // GBK_TO_UNICODE[17875] := 16#7A8A;
   // GBK_TO_UNICODE[17876] := 16#B794;
   // GBK_TO_UNICODE[17877] := 16#7A8B;
   // GBK_TO_UNICODE[17878] := 16#B795;
   // GBK_TO_UNICODE[17879] := 16#7A8C;
   // GBK_TO_UNICODE[17880] := 16#B796;
   // GBK_TO_UNICODE[17881] := 16#7A8E;
   // GBK_TO_UNICODE[17882] := 16#B797;
   // GBK_TO_UNICODE[17883] := 16#7A8F;
   // GBK_TO_UNICODE[17884] := 16#B798;
   // GBK_TO_UNICODE[17885] := 16#7A90;
   // GBK_TO_UNICODE[17886] := 16#B799;
   // GBK_TO_UNICODE[17887] := 16#7A93;
   // GBK_TO_UNICODE[17888] := 16#B79A;
   // GBK_TO_UNICODE[17889] := 16#7A94;
   // GBK_TO_UNICODE[17890] := 16#B79B;
   // GBK_TO_UNICODE[17891] := 16#7A99;
   // GBK_TO_UNICODE[17892] := 16#B79C;
   // GBK_TO_UNICODE[17893] := 16#7A9A;
   // GBK_TO_UNICODE[17894] := 16#B79D;
   // GBK_TO_UNICODE[17895] := 16#7A9B;
   // GBK_TO_UNICODE[17896] := 16#B79E;
   // GBK_TO_UNICODE[17897] := 16#7A9E;
   // GBK_TO_UNICODE[17898] := 16#B79F;
   // GBK_TO_UNICODE[17899] := 16#7AA1;
   // GBK_TO_UNICODE[17900] := 16#B7A0;
   // GBK_TO_UNICODE[17901] := 16#7AA2;
   // GBK_TO_UNICODE[17902] := 16#B7A1;
   // GBK_TO_UNICODE[17903] := 16#8D30;
   // GBK_TO_UNICODE[17904] := 16#B7A2;
   // GBK_TO_UNICODE[17905] := 16#53D1;
   // GBK_TO_UNICODE[17906] := 16#B7A3;
   // GBK_TO_UNICODE[17907] := 16#7F5A;
   // GBK_TO_UNICODE[17908] := 16#B7A4;
   // GBK_TO_UNICODE[17909] := 16#7B4F;
   // GBK_TO_UNICODE[17910] := 16#B7A5;
   // GBK_TO_UNICODE[17911] := 16#4F10;
   // GBK_TO_UNICODE[17912] := 16#B7A6;
   // GBK_TO_UNICODE[17913] := 16#4E4F;
   // GBK_TO_UNICODE[17914] := 16#B7A7;
   // GBK_TO_UNICODE[17915] := 16#9600;
   // GBK_TO_UNICODE[17916] := 16#B7A8;
   // GBK_TO_UNICODE[17917] := 16#6CD5;
   // GBK_TO_UNICODE[17918] := 16#B7A9;
   // GBK_TO_UNICODE[17919] := 16#73D0;
   // GBK_TO_UNICODE[17920] := 16#B7AA;
   // GBK_TO_UNICODE[17921] := 16#85E9;
   // GBK_TO_UNICODE[17922] := 16#B7AB;
   // GBK_TO_UNICODE[17923] := 16#5E06;
   // GBK_TO_UNICODE[17924] := 16#B7AC;
   // GBK_TO_UNICODE[17925] := 16#756A;
   // GBK_TO_UNICODE[17926] := 16#B7AD;
   // GBK_TO_UNICODE[17927] := 16#7FFB;
   // GBK_TO_UNICODE[17928] := 16#B7AE;
   // GBK_TO_UNICODE[17929] := 16#6A0A;
   // GBK_TO_UNICODE[17930] := 16#B7AF;
   // GBK_TO_UNICODE[17931] := 16#77FE;
   // GBK_TO_UNICODE[17932] := 16#B7B0;
   // GBK_TO_UNICODE[17933] := 16#9492;
   // GBK_TO_UNICODE[17934] := 16#B7B1;
   // GBK_TO_UNICODE[17935] := 16#7E41;
   // GBK_TO_UNICODE[17936] := 16#B7B2;
   // GBK_TO_UNICODE[17937] := 16#51E1;
   // GBK_TO_UNICODE[17938] := 16#B7B3;
   // GBK_TO_UNICODE[17939] := 16#70E6;
   // GBK_TO_UNICODE[17940] := 16#B7B4;
   // GBK_TO_UNICODE[17941] := 16#53CD;
   // GBK_TO_UNICODE[17942] := 16#B7B5;
   // GBK_TO_UNICODE[17943] := 16#8FD4;
   // GBK_TO_UNICODE[17944] := 16#B7B6;
   // GBK_TO_UNICODE[17945] := 16#8303;
   // GBK_TO_UNICODE[17946] := 16#B7B7;
   // GBK_TO_UNICODE[17947] := 16#8D29;
   // GBK_TO_UNICODE[17948] := 16#B7B8;
   // GBK_TO_UNICODE[17949] := 16#72AF;
   // GBK_TO_UNICODE[17950] := 16#B7B9;
   // GBK_TO_UNICODE[17951] := 16#996D;
   // GBK_TO_UNICODE[17952] := 16#B7BA;
   // GBK_TO_UNICODE[17953] := 16#6CDB;
   // GBK_TO_UNICODE[17954] := 16#B7BB;
   // GBK_TO_UNICODE[17955] := 16#574A;
   // GBK_TO_UNICODE[17956] := 16#B7BC;
   // GBK_TO_UNICODE[17957] := 16#82B3;
   // GBK_TO_UNICODE[17958] := 16#B7BD;
   // GBK_TO_UNICODE[17959] := 16#65B9;
   // GBK_TO_UNICODE[17960] := 16#B7BE;
   // GBK_TO_UNICODE[17961] := 16#80AA;
   // GBK_TO_UNICODE[17962] := 16#B7BF;
   // GBK_TO_UNICODE[17963] := 16#623F;
   // GBK_TO_UNICODE[17964] := 16#B7C0;
   // GBK_TO_UNICODE[17965] := 16#9632;
   // GBK_TO_UNICODE[17966] := 16#B7C1;
   // GBK_TO_UNICODE[17967] := 16#59A8;
   // GBK_TO_UNICODE[17968] := 16#B7C2;
   // GBK_TO_UNICODE[17969] := 16#4EFF;
   // GBK_TO_UNICODE[17970] := 16#B7C3;
   // GBK_TO_UNICODE[17971] := 16#8BBF;
   // GBK_TO_UNICODE[17972] := 16#B7C4;
   // GBK_TO_UNICODE[17973] := 16#7EBA;
   // GBK_TO_UNICODE[17974] := 16#B7C5;
   // GBK_TO_UNICODE[17975] := 16#653E;
   // GBK_TO_UNICODE[17976] := 16#B7C6;
   // GBK_TO_UNICODE[17977] := 16#83F2;
   // GBK_TO_UNICODE[17978] := 16#B7C7;
   // GBK_TO_UNICODE[17979] := 16#975E;
   // GBK_TO_UNICODE[17980] := 16#B7C8;
   // GBK_TO_UNICODE[17981] := 16#5561;
   // GBK_TO_UNICODE[17982] := 16#B7C9;
   // GBK_TO_UNICODE[17983] := 16#98DE;
   // GBK_TO_UNICODE[17984] := 16#B7CA;
   // GBK_TO_UNICODE[17985] := 16#80A5;
   // GBK_TO_UNICODE[17986] := 16#B7CB;
   // GBK_TO_UNICODE[17987] := 16#532A;
   // GBK_TO_UNICODE[17988] := 16#B7CC;
   // GBK_TO_UNICODE[17989] := 16#8BFD;
   // GBK_TO_UNICODE[17990] := 16#B7CD;
   // GBK_TO_UNICODE[17991] := 16#5420;
   // GBK_TO_UNICODE[17992] := 16#B7CE;
   // GBK_TO_UNICODE[17993] := 16#80BA;
   // GBK_TO_UNICODE[17994] := 16#B7CF;
   // GBK_TO_UNICODE[17995] := 16#5E9F;
   // GBK_TO_UNICODE[17996] := 16#B7D0;
   // GBK_TO_UNICODE[17997] := 16#6CB8;
   // GBK_TO_UNICODE[17998] := 16#B7D1;
   // GBK_TO_UNICODE[17999] := 16#8D39;
   // GBK_TO_UNICODE[18000] := 16#B7D2;
   // GBK_TO_UNICODE[18001] := 16#82AC;
   // GBK_TO_UNICODE[18002] := 16#B7D3;
   // GBK_TO_UNICODE[18003] := 16#915A;
   // GBK_TO_UNICODE[18004] := 16#B7D4;
   // GBK_TO_UNICODE[18005] := 16#5429;
   // GBK_TO_UNICODE[18006] := 16#B7D5;
   // GBK_TO_UNICODE[18007] := 16#6C1B;
   // GBK_TO_UNICODE[18008] := 16#B7D6;
   // GBK_TO_UNICODE[18009] := 16#5206;
   // GBK_TO_UNICODE[18010] := 16#B7D7;
   // GBK_TO_UNICODE[18011] := 16#7EB7;
   // GBK_TO_UNICODE[18012] := 16#B7D8;
   // GBK_TO_UNICODE[18013] := 16#575F;
   // GBK_TO_UNICODE[18014] := 16#B7D9;
   // GBK_TO_UNICODE[18015] := 16#711A;
   // GBK_TO_UNICODE[18016] := 16#B7DA;
   // GBK_TO_UNICODE[18017] := 16#6C7E;
   // GBK_TO_UNICODE[18018] := 16#B7DB;
   // GBK_TO_UNICODE[18019] := 16#7C89;
   // GBK_TO_UNICODE[18020] := 16#B7DC;
   // GBK_TO_UNICODE[18021] := 16#594B;
   // GBK_TO_UNICODE[18022] := 16#B7DD;
   // GBK_TO_UNICODE[18023] := 16#4EFD;
   // GBK_TO_UNICODE[18024] := 16#B7DE;
   // GBK_TO_UNICODE[18025] := 16#5FFF;
   // GBK_TO_UNICODE[18026] := 16#B7DF;
   // GBK_TO_UNICODE[18027] := 16#6124;
   // GBK_TO_UNICODE[18028] := 16#B7E0;
   // GBK_TO_UNICODE[18029] := 16#7CAA;
   // GBK_TO_UNICODE[18030] := 16#B7E1;
   // GBK_TO_UNICODE[18031] := 16#4E30;
   // GBK_TO_UNICODE[18032] := 16#B7E2;
   // GBK_TO_UNICODE[18033] := 16#5C01;
   // GBK_TO_UNICODE[18034] := 16#B7E3;
   // GBK_TO_UNICODE[18035] := 16#67AB;
   // GBK_TO_UNICODE[18036] := 16#B7E4;
   // GBK_TO_UNICODE[18037] := 16#8702;
   // GBK_TO_UNICODE[18038] := 16#B7E5;
   // GBK_TO_UNICODE[18039] := 16#5CF0;
   // GBK_TO_UNICODE[18040] := 16#B7E6;
   // GBK_TO_UNICODE[18041] := 16#950B;
   // GBK_TO_UNICODE[18042] := 16#B7E7;
   // GBK_TO_UNICODE[18043] := 16#98CE;
   // GBK_TO_UNICODE[18044] := 16#B7E8;
   // GBK_TO_UNICODE[18045] := 16#75AF;
   // GBK_TO_UNICODE[18046] := 16#B7E9;
   // GBK_TO_UNICODE[18047] := 16#70FD;
   // GBK_TO_UNICODE[18048] := 16#B7EA;
   // GBK_TO_UNICODE[18049] := 16#9022;
   // GBK_TO_UNICODE[18050] := 16#B7EB;
   // GBK_TO_UNICODE[18051] := 16#51AF;
   // GBK_TO_UNICODE[18052] := 16#B7EC;
   // GBK_TO_UNICODE[18053] := 16#7F1D;
   // GBK_TO_UNICODE[18054] := 16#B7ED;
   // GBK_TO_UNICODE[18055] := 16#8BBD;
   // GBK_TO_UNICODE[18056] := 16#B7EE;
   // GBK_TO_UNICODE[18057] := 16#5949;
   // GBK_TO_UNICODE[18058] := 16#B7EF;
   // GBK_TO_UNICODE[18059] := 16#51E4;
   // GBK_TO_UNICODE[18060] := 16#B7F0;
   // GBK_TO_UNICODE[18061] := 16#4F5B;
   // GBK_TO_UNICODE[18062] := 16#B7F1;
   // GBK_TO_UNICODE[18063] := 16#5426;
   // GBK_TO_UNICODE[18064] := 16#B7F2;
   // GBK_TO_UNICODE[18065] := 16#592B;
   // GBK_TO_UNICODE[18066] := 16#B7F3;
   // GBK_TO_UNICODE[18067] := 16#6577;
   // GBK_TO_UNICODE[18068] := 16#B7F4;
   // GBK_TO_UNICODE[18069] := 16#80A4;
   // GBK_TO_UNICODE[18070] := 16#B7F5;
   // GBK_TO_UNICODE[18071] := 16#5B75;
   // GBK_TO_UNICODE[18072] := 16#B7F6;
   // GBK_TO_UNICODE[18073] := 16#6276;
   // GBK_TO_UNICODE[18074] := 16#B7F7;
   // GBK_TO_UNICODE[18075] := 16#62C2;
   // GBK_TO_UNICODE[18076] := 16#B7F8;
   // GBK_TO_UNICODE[18077] := 16#8F90;
   // GBK_TO_UNICODE[18078] := 16#B7F9;
   // GBK_TO_UNICODE[18079] := 16#5E45;
   // GBK_TO_UNICODE[18080] := 16#B7FA;
   // GBK_TO_UNICODE[18081] := 16#6C1F;
   // GBK_TO_UNICODE[18082] := 16#B7FB;
   // GBK_TO_UNICODE[18083] := 16#7B26;
   // GBK_TO_UNICODE[18084] := 16#B7FC;
   // GBK_TO_UNICODE[18085] := 16#4F0F;
   // GBK_TO_UNICODE[18086] := 16#B7FD;
   // GBK_TO_UNICODE[18087] := 16#4FD8;
   // GBK_TO_UNICODE[18088] := 16#B7FE;
   // GBK_TO_UNICODE[18089] := 16#670D;
   // GBK_TO_UNICODE[18090] := 16#B840;
   // GBK_TO_UNICODE[18091] := 16#7AA3;
   // GBK_TO_UNICODE[18092] := 16#B841;
   // GBK_TO_UNICODE[18093] := 16#7AA4;
   // GBK_TO_UNICODE[18094] := 16#B842;
   // GBK_TO_UNICODE[18095] := 16#7AA7;
   // GBK_TO_UNICODE[18096] := 16#B843;
   // GBK_TO_UNICODE[18097] := 16#7AA9;
   // GBK_TO_UNICODE[18098] := 16#B844;
   // GBK_TO_UNICODE[18099] := 16#7AAA;
   // GBK_TO_UNICODE[18100] := 16#B845;
   // GBK_TO_UNICODE[18101] := 16#7AAB;
   // GBK_TO_UNICODE[18102] := 16#B846;
   // GBK_TO_UNICODE[18103] := 16#7AAE;
   // GBK_TO_UNICODE[18104] := 16#B847;
   // GBK_TO_UNICODE[18105] := 16#7AAF;
   // GBK_TO_UNICODE[18106] := 16#B848;
   // GBK_TO_UNICODE[18107] := 16#7AB0;
   // GBK_TO_UNICODE[18108] := 16#B849;
   // GBK_TO_UNICODE[18109] := 16#7AB1;
   // GBK_TO_UNICODE[18110] := 16#B84A;
   // GBK_TO_UNICODE[18111] := 16#7AB2;
   // GBK_TO_UNICODE[18112] := 16#B84B;
   // GBK_TO_UNICODE[18113] := 16#7AB4;
   // GBK_TO_UNICODE[18114] := 16#B84C;
   // GBK_TO_UNICODE[18115] := 16#7AB5;
   // GBK_TO_UNICODE[18116] := 16#B84D;
   // GBK_TO_UNICODE[18117] := 16#7AB6;
   // GBK_TO_UNICODE[18118] := 16#B84E;
   // GBK_TO_UNICODE[18119] := 16#7AB7;
   // GBK_TO_UNICODE[18120] := 16#B84F;
   // GBK_TO_UNICODE[18121] := 16#7AB8;
   // GBK_TO_UNICODE[18122] := 16#B850;
   // GBK_TO_UNICODE[18123] := 16#7AB9;
   // GBK_TO_UNICODE[18124] := 16#B851;
   // GBK_TO_UNICODE[18125] := 16#7ABA;
   // GBK_TO_UNICODE[18126] := 16#B852;
   // GBK_TO_UNICODE[18127] := 16#7ABB;
   // GBK_TO_UNICODE[18128] := 16#B853;
   // GBK_TO_UNICODE[18129] := 16#7ABC;
   // GBK_TO_UNICODE[18130] := 16#B854;
   // GBK_TO_UNICODE[18131] := 16#7ABD;
   // GBK_TO_UNICODE[18132] := 16#B855;
   // GBK_TO_UNICODE[18133] := 16#7ABE;
   // GBK_TO_UNICODE[18134] := 16#B856;
   // GBK_TO_UNICODE[18135] := 16#7AC0;
   // GBK_TO_UNICODE[18136] := 16#B857;
   // GBK_TO_UNICODE[18137] := 16#7AC1;
   // GBK_TO_UNICODE[18138] := 16#B858;
   // GBK_TO_UNICODE[18139] := 16#7AC2;
   // GBK_TO_UNICODE[18140] := 16#B859;
   // GBK_TO_UNICODE[18141] := 16#7AC3;
   // GBK_TO_UNICODE[18142] := 16#B85A;
   // GBK_TO_UNICODE[18143] := 16#7AC4;
   // GBK_TO_UNICODE[18144] := 16#B85B;
   // GBK_TO_UNICODE[18145] := 16#7AC5;
   // GBK_TO_UNICODE[18146] := 16#B85C;
   // GBK_TO_UNICODE[18147] := 16#7AC6;
   // GBK_TO_UNICODE[18148] := 16#B85D;
   // GBK_TO_UNICODE[18149] := 16#7AC7;
   // GBK_TO_UNICODE[18150] := 16#B85E;
   // GBK_TO_UNICODE[18151] := 16#7AC8;
   // GBK_TO_UNICODE[18152] := 16#B85F;
   // GBK_TO_UNICODE[18153] := 16#7AC9;
   // GBK_TO_UNICODE[18154] := 16#B860;
   // GBK_TO_UNICODE[18155] := 16#7ACA;
   // GBK_TO_UNICODE[18156] := 16#B861;
   // GBK_TO_UNICODE[18157] := 16#7ACC;
   // GBK_TO_UNICODE[18158] := 16#B862;
   // GBK_TO_UNICODE[18159] := 16#7ACD;
   // GBK_TO_UNICODE[18160] := 16#B863;
   // GBK_TO_UNICODE[18161] := 16#7ACE;
   // GBK_TO_UNICODE[18162] := 16#B864;
   // GBK_TO_UNICODE[18163] := 16#7ACF;
   // GBK_TO_UNICODE[18164] := 16#B865;
   // GBK_TO_UNICODE[18165] := 16#7AD0;
   // GBK_TO_UNICODE[18166] := 16#B866;
   // GBK_TO_UNICODE[18167] := 16#7AD1;
   // GBK_TO_UNICODE[18168] := 16#B867;
   // GBK_TO_UNICODE[18169] := 16#7AD2;
   // GBK_TO_UNICODE[18170] := 16#B868;
   // GBK_TO_UNICODE[18171] := 16#7AD3;
   // GBK_TO_UNICODE[18172] := 16#B869;
   // GBK_TO_UNICODE[18173] := 16#7AD4;
   // GBK_TO_UNICODE[18174] := 16#B86A;
   // GBK_TO_UNICODE[18175] := 16#7AD5;
   // GBK_TO_UNICODE[18176] := 16#B86B;
   // GBK_TO_UNICODE[18177] := 16#7AD7;
   // GBK_TO_UNICODE[18178] := 16#B86C;
   // GBK_TO_UNICODE[18179] := 16#7AD8;
   // GBK_TO_UNICODE[18180] := 16#B86D;
   // GBK_TO_UNICODE[18181] := 16#7ADA;
   // GBK_TO_UNICODE[18182] := 16#B86E;
   // GBK_TO_UNICODE[18183] := 16#7ADB;
   // GBK_TO_UNICODE[18184] := 16#B86F;
   // GBK_TO_UNICODE[18185] := 16#7ADC;
   // GBK_TO_UNICODE[18186] := 16#B870;
   // GBK_TO_UNICODE[18187] := 16#7ADD;
   // GBK_TO_UNICODE[18188] := 16#B871;
   // GBK_TO_UNICODE[18189] := 16#7AE1;
   // GBK_TO_UNICODE[18190] := 16#B872;
   // GBK_TO_UNICODE[18191] := 16#7AE2;
   // GBK_TO_UNICODE[18192] := 16#B873;
   // GBK_TO_UNICODE[18193] := 16#7AE4;
   // GBK_TO_UNICODE[18194] := 16#B874;
   // GBK_TO_UNICODE[18195] := 16#7AE7;
   // GBK_TO_UNICODE[18196] := 16#B875;
   // GBK_TO_UNICODE[18197] := 16#7AE8;
   // GBK_TO_UNICODE[18198] := 16#B876;
   // GBK_TO_UNICODE[18199] := 16#7AE9;
   // GBK_TO_UNICODE[18200] := 16#B877;
   // GBK_TO_UNICODE[18201] := 16#7AEA;
   // GBK_TO_UNICODE[18202] := 16#B878;
   // GBK_TO_UNICODE[18203] := 16#7AEB;
   // GBK_TO_UNICODE[18204] := 16#B879;
   // GBK_TO_UNICODE[18205] := 16#7AEC;
   // GBK_TO_UNICODE[18206] := 16#B87A;
   // GBK_TO_UNICODE[18207] := 16#7AEE;
   // GBK_TO_UNICODE[18208] := 16#B87B;
   // GBK_TO_UNICODE[18209] := 16#7AF0;
   // GBK_TO_UNICODE[18210] := 16#B87C;
   // GBK_TO_UNICODE[18211] := 16#7AF1;
   // GBK_TO_UNICODE[18212] := 16#B87D;
   // GBK_TO_UNICODE[18213] := 16#7AF2;
   // GBK_TO_UNICODE[18214] := 16#B87E;
   // GBK_TO_UNICODE[18215] := 16#7AF3;
   // GBK_TO_UNICODE[18216] := 16#B880;
   // GBK_TO_UNICODE[18217] := 16#7AF4;
   // GBK_TO_UNICODE[18218] := 16#B881;
   // GBK_TO_UNICODE[18219] := 16#7AF5;
   // GBK_TO_UNICODE[18220] := 16#B882;
   // GBK_TO_UNICODE[18221] := 16#7AF6;
   // GBK_TO_UNICODE[18222] := 16#B883;
   // GBK_TO_UNICODE[18223] := 16#7AF7;
   // GBK_TO_UNICODE[18224] := 16#B884;
   // GBK_TO_UNICODE[18225] := 16#7AF8;
   // GBK_TO_UNICODE[18226] := 16#B885;
   // GBK_TO_UNICODE[18227] := 16#7AFB;
   // GBK_TO_UNICODE[18228] := 16#B886;
   // GBK_TO_UNICODE[18229] := 16#7AFC;
   // GBK_TO_UNICODE[18230] := 16#B887;
   // GBK_TO_UNICODE[18231] := 16#7AFE;
   // GBK_TO_UNICODE[18232] := 16#B888;
   // GBK_TO_UNICODE[18233] := 16#7B00;
   // GBK_TO_UNICODE[18234] := 16#B889;
   // GBK_TO_UNICODE[18235] := 16#7B01;
   // GBK_TO_UNICODE[18236] := 16#B88A;
   // GBK_TO_UNICODE[18237] := 16#7B02;
   // GBK_TO_UNICODE[18238] := 16#B88B;
   // GBK_TO_UNICODE[18239] := 16#7B05;
   // GBK_TO_UNICODE[18240] := 16#B88C;
   // GBK_TO_UNICODE[18241] := 16#7B07;
   // GBK_TO_UNICODE[18242] := 16#B88D;
   // GBK_TO_UNICODE[18243] := 16#7B09;
   // GBK_TO_UNICODE[18244] := 16#B88E;
   // GBK_TO_UNICODE[18245] := 16#7B0C;
   // GBK_TO_UNICODE[18246] := 16#B88F;
   // GBK_TO_UNICODE[18247] := 16#7B0D;
   // GBK_TO_UNICODE[18248] := 16#B890;
   // GBK_TO_UNICODE[18249] := 16#7B0E;
   // GBK_TO_UNICODE[18250] := 16#B891;
   // GBK_TO_UNICODE[18251] := 16#7B10;
   // GBK_TO_UNICODE[18252] := 16#B892;
   // GBK_TO_UNICODE[18253] := 16#7B12;
   // GBK_TO_UNICODE[18254] := 16#B893;
   // GBK_TO_UNICODE[18255] := 16#7B13;
   // GBK_TO_UNICODE[18256] := 16#B894;
   // GBK_TO_UNICODE[18257] := 16#7B16;
   // GBK_TO_UNICODE[18258] := 16#B895;
   // GBK_TO_UNICODE[18259] := 16#7B17;
   // GBK_TO_UNICODE[18260] := 16#B896;
   // GBK_TO_UNICODE[18261] := 16#7B18;
   // GBK_TO_UNICODE[18262] := 16#B897;
   // GBK_TO_UNICODE[18263] := 16#7B1A;
   // GBK_TO_UNICODE[18264] := 16#B898;
   // GBK_TO_UNICODE[18265] := 16#7B1C;
   // GBK_TO_UNICODE[18266] := 16#B899;
   // GBK_TO_UNICODE[18267] := 16#7B1D;
   // GBK_TO_UNICODE[18268] := 16#B89A;
   // GBK_TO_UNICODE[18269] := 16#7B1F;
   // GBK_TO_UNICODE[18270] := 16#B89B;
   // GBK_TO_UNICODE[18271] := 16#7B21;
   // GBK_TO_UNICODE[18272] := 16#B89C;
   // GBK_TO_UNICODE[18273] := 16#7B22;
   // GBK_TO_UNICODE[18274] := 16#B89D;
   // GBK_TO_UNICODE[18275] := 16#7B23;
   // GBK_TO_UNICODE[18276] := 16#B89E;
   // GBK_TO_UNICODE[18277] := 16#7B27;
   // GBK_TO_UNICODE[18278] := 16#B89F;
   // GBK_TO_UNICODE[18279] := 16#7B29;
   // GBK_TO_UNICODE[18280] := 16#B8A0;
   // GBK_TO_UNICODE[18281] := 16#7B2D;
   // GBK_TO_UNICODE[18282] := 16#B8A1;
   // GBK_TO_UNICODE[18283] := 16#6D6E;
   // GBK_TO_UNICODE[18284] := 16#B8A2;
   // GBK_TO_UNICODE[18285] := 16#6DAA;
   // GBK_TO_UNICODE[18286] := 16#B8A3;
   // GBK_TO_UNICODE[18287] := 16#798F;
   // GBK_TO_UNICODE[18288] := 16#B8A4;
   // GBK_TO_UNICODE[18289] := 16#88B1;
   // GBK_TO_UNICODE[18290] := 16#B8A5;
   // GBK_TO_UNICODE[18291] := 16#5F17;
   // GBK_TO_UNICODE[18292] := 16#B8A6;
   // GBK_TO_UNICODE[18293] := 16#752B;
   // GBK_TO_UNICODE[18294] := 16#B8A7;
   // GBK_TO_UNICODE[18295] := 16#629A;
   // GBK_TO_UNICODE[18296] := 16#B8A8;
   // GBK_TO_UNICODE[18297] := 16#8F85;
   // GBK_TO_UNICODE[18298] := 16#B8A9;
   // GBK_TO_UNICODE[18299] := 16#4FEF;
   // GBK_TO_UNICODE[18300] := 16#B8AA;
   // GBK_TO_UNICODE[18301] := 16#91DC;
   // GBK_TO_UNICODE[18302] := 16#B8AB;
   // GBK_TO_UNICODE[18303] := 16#65A7;
   // GBK_TO_UNICODE[18304] := 16#B8AC;
   // GBK_TO_UNICODE[18305] := 16#812F;
   // GBK_TO_UNICODE[18306] := 16#B8AD;
   // GBK_TO_UNICODE[18307] := 16#8151;
   // GBK_TO_UNICODE[18308] := 16#B8AE;
   // GBK_TO_UNICODE[18309] := 16#5E9C;
   // GBK_TO_UNICODE[18310] := 16#B8AF;
   // GBK_TO_UNICODE[18311] := 16#8150;
   // GBK_TO_UNICODE[18312] := 16#B8B0;
   // GBK_TO_UNICODE[18313] := 16#8D74;
   // GBK_TO_UNICODE[18314] := 16#B8B1;
   // GBK_TO_UNICODE[18315] := 16#526F;
   // GBK_TO_UNICODE[18316] := 16#B8B2;
   // GBK_TO_UNICODE[18317] := 16#8986;
   // GBK_TO_UNICODE[18318] := 16#B8B3;
   // GBK_TO_UNICODE[18319] := 16#8D4B;
   // GBK_TO_UNICODE[18320] := 16#B8B4;
   // GBK_TO_UNICODE[18321] := 16#590D;
   // GBK_TO_UNICODE[18322] := 16#B8B5;
   // GBK_TO_UNICODE[18323] := 16#5085;
   // GBK_TO_UNICODE[18324] := 16#B8B6;
   // GBK_TO_UNICODE[18325] := 16#4ED8;
   // GBK_TO_UNICODE[18326] := 16#B8B7;
   // GBK_TO_UNICODE[18327] := 16#961C;
   // GBK_TO_UNICODE[18328] := 16#B8B8;
   // GBK_TO_UNICODE[18329] := 16#7236;
   // GBK_TO_UNICODE[18330] := 16#B8B9;
   // GBK_TO_UNICODE[18331] := 16#8179;
   // GBK_TO_UNICODE[18332] := 16#B8BA;
   // GBK_TO_UNICODE[18333] := 16#8D1F;
   // GBK_TO_UNICODE[18334] := 16#B8BB;
   // GBK_TO_UNICODE[18335] := 16#5BCC;
   // GBK_TO_UNICODE[18336] := 16#B8BC;
   // GBK_TO_UNICODE[18337] := 16#8BA3;
   // GBK_TO_UNICODE[18338] := 16#B8BD;
   // GBK_TO_UNICODE[18339] := 16#9644;
   // GBK_TO_UNICODE[18340] := 16#B8BE;
   // GBK_TO_UNICODE[18341] := 16#5987;
   // GBK_TO_UNICODE[18342] := 16#B8BF;
   // GBK_TO_UNICODE[18343] := 16#7F1A;
   // GBK_TO_UNICODE[18344] := 16#B8C0;
   // GBK_TO_UNICODE[18345] := 16#5490;
   // GBK_TO_UNICODE[18346] := 16#B8C1;
   // GBK_TO_UNICODE[18347] := 16#5676;
   // GBK_TO_UNICODE[18348] := 16#B8C2;
   // GBK_TO_UNICODE[18349] := 16#560E;
   // GBK_TO_UNICODE[18350] := 16#B8C3;
   // GBK_TO_UNICODE[18351] := 16#8BE5;
   // GBK_TO_UNICODE[18352] := 16#B8C4;
   // GBK_TO_UNICODE[18353] := 16#6539;
   // GBK_TO_UNICODE[18354] := 16#B8C5;
   // GBK_TO_UNICODE[18355] := 16#6982;
   // GBK_TO_UNICODE[18356] := 16#B8C6;
   // GBK_TO_UNICODE[18357] := 16#9499;
   // GBK_TO_UNICODE[18358] := 16#B8C7;
   // GBK_TO_UNICODE[18359] := 16#76D6;
   // GBK_TO_UNICODE[18360] := 16#B8C8;
   // GBK_TO_UNICODE[18361] := 16#6E89;
   // GBK_TO_UNICODE[18362] := 16#B8C9;
   // GBK_TO_UNICODE[18363] := 16#5E72;
   // GBK_TO_UNICODE[18364] := 16#B8CA;
   // GBK_TO_UNICODE[18365] := 16#7518;
   // GBK_TO_UNICODE[18366] := 16#B8CB;
   // GBK_TO_UNICODE[18367] := 16#6746;
   // GBK_TO_UNICODE[18368] := 16#B8CC;
   // GBK_TO_UNICODE[18369] := 16#67D1;
   // GBK_TO_UNICODE[18370] := 16#B8CD;
   // GBK_TO_UNICODE[18371] := 16#7AFF;
   // GBK_TO_UNICODE[18372] := 16#B8CE;
   // GBK_TO_UNICODE[18373] := 16#809D;
   // GBK_TO_UNICODE[18374] := 16#B8CF;
   // GBK_TO_UNICODE[18375] := 16#8D76;
   // GBK_TO_UNICODE[18376] := 16#B8D0;
   // GBK_TO_UNICODE[18377] := 16#611F;
   // GBK_TO_UNICODE[18378] := 16#B8D1;
   // GBK_TO_UNICODE[18379] := 16#79C6;
   // GBK_TO_UNICODE[18380] := 16#B8D2;
   // GBK_TO_UNICODE[18381] := 16#6562;
   // GBK_TO_UNICODE[18382] := 16#B8D3;
   // GBK_TO_UNICODE[18383] := 16#8D63;
   // GBK_TO_UNICODE[18384] := 16#B8D4;
   // GBK_TO_UNICODE[18385] := 16#5188;
   // GBK_TO_UNICODE[18386] := 16#B8D5;
   // GBK_TO_UNICODE[18387] := 16#521A;
   // GBK_TO_UNICODE[18388] := 16#B8D6;
   // GBK_TO_UNICODE[18389] := 16#94A2;
   // GBK_TO_UNICODE[18390] := 16#B8D7;
   // GBK_TO_UNICODE[18391] := 16#7F38;
   // GBK_TO_UNICODE[18392] := 16#B8D8;
   // GBK_TO_UNICODE[18393] := 16#809B;
   // GBK_TO_UNICODE[18394] := 16#B8D9;
   // GBK_TO_UNICODE[18395] := 16#7EB2;
   // GBK_TO_UNICODE[18396] := 16#B8DA;
   // GBK_TO_UNICODE[18397] := 16#5C97;
   // GBK_TO_UNICODE[18398] := 16#B8DB;
   // GBK_TO_UNICODE[18399] := 16#6E2F;
   // GBK_TO_UNICODE[18400] := 16#B8DC;
   // GBK_TO_UNICODE[18401] := 16#6760;
   // GBK_TO_UNICODE[18402] := 16#B8DD;
   // GBK_TO_UNICODE[18403] := 16#7BD9;
   // GBK_TO_UNICODE[18404] := 16#B8DE;
   // GBK_TO_UNICODE[18405] := 16#768B;
   // GBK_TO_UNICODE[18406] := 16#B8DF;
   // GBK_TO_UNICODE[18407] := 16#9AD8;
   // GBK_TO_UNICODE[18408] := 16#B8E0;
   // GBK_TO_UNICODE[18409] := 16#818F;
   // GBK_TO_UNICODE[18410] := 16#B8E1;
   // GBK_TO_UNICODE[18411] := 16#7F94;
   // GBK_TO_UNICODE[18412] := 16#B8E2;
   // GBK_TO_UNICODE[18413] := 16#7CD5;
   // GBK_TO_UNICODE[18414] := 16#B8E3;
   // GBK_TO_UNICODE[18415] := 16#641E;
   // GBK_TO_UNICODE[18416] := 16#B8E4;
   // GBK_TO_UNICODE[18417] := 16#9550;
   // GBK_TO_UNICODE[18418] := 16#B8E5;
   // GBK_TO_UNICODE[18419] := 16#7A3F;
   // GBK_TO_UNICODE[18420] := 16#B8E6;
   // GBK_TO_UNICODE[18421] := 16#544A;
   // GBK_TO_UNICODE[18422] := 16#B8E7;
   // GBK_TO_UNICODE[18423] := 16#54E5;
   // GBK_TO_UNICODE[18424] := 16#B8E8;
   // GBK_TO_UNICODE[18425] := 16#6B4C;
   // GBK_TO_UNICODE[18426] := 16#B8E9;
   // GBK_TO_UNICODE[18427] := 16#6401;
   // GBK_TO_UNICODE[18428] := 16#B8EA;
   // GBK_TO_UNICODE[18429] := 16#6208;
   // GBK_TO_UNICODE[18430] := 16#B8EB;
   // GBK_TO_UNICODE[18431] := 16#9E3D;
   // GBK_TO_UNICODE[18432] := 16#B8EC;
   // GBK_TO_UNICODE[18433] := 16#80F3;
   // GBK_TO_UNICODE[18434] := 16#B8ED;
   // GBK_TO_UNICODE[18435] := 16#7599;
   // GBK_TO_UNICODE[18436] := 16#B8EE;
   // GBK_TO_UNICODE[18437] := 16#5272;
   // GBK_TO_UNICODE[18438] := 16#B8EF;
   // GBK_TO_UNICODE[18439] := 16#9769;
   // GBK_TO_UNICODE[18440] := 16#B8F0;
   // GBK_TO_UNICODE[18441] := 16#845B;
   // GBK_TO_UNICODE[18442] := 16#B8F1;
   // GBK_TO_UNICODE[18443] := 16#683C;
   // GBK_TO_UNICODE[18444] := 16#B8F2;
   // GBK_TO_UNICODE[18445] := 16#86E4;
   // GBK_TO_UNICODE[18446] := 16#B8F3;
   // GBK_TO_UNICODE[18447] := 16#9601;
   // GBK_TO_UNICODE[18448] := 16#B8F4;
   // GBK_TO_UNICODE[18449] := 16#9694;
   // GBK_TO_UNICODE[18450] := 16#B8F5;
   // GBK_TO_UNICODE[18451] := 16#94EC;
   // GBK_TO_UNICODE[18452] := 16#B8F6;
   // GBK_TO_UNICODE[18453] := 16#4E2A;
   // GBK_TO_UNICODE[18454] := 16#B8F7;
   // GBK_TO_UNICODE[18455] := 16#5404;
   // GBK_TO_UNICODE[18456] := 16#B8F8;
   // GBK_TO_UNICODE[18457] := 16#7ED9;
   // GBK_TO_UNICODE[18458] := 16#B8F9;
   // GBK_TO_UNICODE[18459] := 16#6839;
   // GBK_TO_UNICODE[18460] := 16#B8FA;
   // GBK_TO_UNICODE[18461] := 16#8DDF;
   // GBK_TO_UNICODE[18462] := 16#B8FB;
   // GBK_TO_UNICODE[18463] := 16#8015;
   // GBK_TO_UNICODE[18464] := 16#B8FC;
   // GBK_TO_UNICODE[18465] := 16#66F4;
   // GBK_TO_UNICODE[18466] := 16#B8FD;
   // GBK_TO_UNICODE[18467] := 16#5E9A;
   // GBK_TO_UNICODE[18468] := 16#B8FE;
   // GBK_TO_UNICODE[18469] := 16#7FB9;
   // GBK_TO_UNICODE[18470] := 16#B940;
   // GBK_TO_UNICODE[18471] := 16#7B2F;
   // GBK_TO_UNICODE[18472] := 16#B941;
   // GBK_TO_UNICODE[18473] := 16#7B30;
   // GBK_TO_UNICODE[18474] := 16#B942;
   // GBK_TO_UNICODE[18475] := 16#7B32;
   // GBK_TO_UNICODE[18476] := 16#B943;
   // GBK_TO_UNICODE[18477] := 16#7B34;
   // GBK_TO_UNICODE[18478] := 16#B944;
   // GBK_TO_UNICODE[18479] := 16#7B35;
   // GBK_TO_UNICODE[18480] := 16#B945;
   // GBK_TO_UNICODE[18481] := 16#7B36;
   // GBK_TO_UNICODE[18482] := 16#B946;
   // GBK_TO_UNICODE[18483] := 16#7B37;
   // GBK_TO_UNICODE[18484] := 16#B947;
   // GBK_TO_UNICODE[18485] := 16#7B39;
   // GBK_TO_UNICODE[18486] := 16#B948;
   // GBK_TO_UNICODE[18487] := 16#7B3B;
   // GBK_TO_UNICODE[18488] := 16#B949;
   // GBK_TO_UNICODE[18489] := 16#7B3D;
   // GBK_TO_UNICODE[18490] := 16#B94A;
   // GBK_TO_UNICODE[18491] := 16#7B3F;
   // GBK_TO_UNICODE[18492] := 16#B94B;
   // GBK_TO_UNICODE[18493] := 16#7B40;
   // GBK_TO_UNICODE[18494] := 16#B94C;
   // GBK_TO_UNICODE[18495] := 16#7B41;
   // GBK_TO_UNICODE[18496] := 16#B94D;
   // GBK_TO_UNICODE[18497] := 16#7B42;
   // GBK_TO_UNICODE[18498] := 16#B94E;
   // GBK_TO_UNICODE[18499] := 16#7B43;
   // GBK_TO_UNICODE[18500] := 16#B94F;
   // GBK_TO_UNICODE[18501] := 16#7B44;
   // GBK_TO_UNICODE[18502] := 16#B950;
   // GBK_TO_UNICODE[18503] := 16#7B46;
   // GBK_TO_UNICODE[18504] := 16#B951;
   // GBK_TO_UNICODE[18505] := 16#7B48;
   // GBK_TO_UNICODE[18506] := 16#B952;
   // GBK_TO_UNICODE[18507] := 16#7B4A;
   // GBK_TO_UNICODE[18508] := 16#B953;
   // GBK_TO_UNICODE[18509] := 16#7B4D;
   // GBK_TO_UNICODE[18510] := 16#B954;
   // GBK_TO_UNICODE[18511] := 16#7B4E;
   // GBK_TO_UNICODE[18512] := 16#B955;
   // GBK_TO_UNICODE[18513] := 16#7B53;
   // GBK_TO_UNICODE[18514] := 16#B956;
   // GBK_TO_UNICODE[18515] := 16#7B55;
   // GBK_TO_UNICODE[18516] := 16#B957;
   // GBK_TO_UNICODE[18517] := 16#7B57;
   // GBK_TO_UNICODE[18518] := 16#B958;
   // GBK_TO_UNICODE[18519] := 16#7B59;
   // GBK_TO_UNICODE[18520] := 16#B959;
   // GBK_TO_UNICODE[18521] := 16#7B5C;
   // GBK_TO_UNICODE[18522] := 16#B95A;
   // GBK_TO_UNICODE[18523] := 16#7B5E;
   // GBK_TO_UNICODE[18524] := 16#B95B;
   // GBK_TO_UNICODE[18525] := 16#7B5F;
   // GBK_TO_UNICODE[18526] := 16#B95C;
   // GBK_TO_UNICODE[18527] := 16#7B61;
   // GBK_TO_UNICODE[18528] := 16#B95D;
   // GBK_TO_UNICODE[18529] := 16#7B63;
   // GBK_TO_UNICODE[18530] := 16#B95E;
   // GBK_TO_UNICODE[18531] := 16#7B64;
   // GBK_TO_UNICODE[18532] := 16#B95F;
   // GBK_TO_UNICODE[18533] := 16#7B65;
   // GBK_TO_UNICODE[18534] := 16#B960;
   // GBK_TO_UNICODE[18535] := 16#7B66;
   // GBK_TO_UNICODE[18536] := 16#B961;
   // GBK_TO_UNICODE[18537] := 16#7B67;
   // GBK_TO_UNICODE[18538] := 16#B962;
   // GBK_TO_UNICODE[18539] := 16#7B68;
   // GBK_TO_UNICODE[18540] := 16#B963;
   // GBK_TO_UNICODE[18541] := 16#7B69;
   // GBK_TO_UNICODE[18542] := 16#B964;
   // GBK_TO_UNICODE[18543] := 16#7B6A;
   // GBK_TO_UNICODE[18544] := 16#B965;
   // GBK_TO_UNICODE[18545] := 16#7B6B;
   // GBK_TO_UNICODE[18546] := 16#B966;
   // GBK_TO_UNICODE[18547] := 16#7B6C;
   // GBK_TO_UNICODE[18548] := 16#B967;
   // GBK_TO_UNICODE[18549] := 16#7B6D;
   // GBK_TO_UNICODE[18550] := 16#B968;
   // GBK_TO_UNICODE[18551] := 16#7B6F;
   // GBK_TO_UNICODE[18552] := 16#B969;
   // GBK_TO_UNICODE[18553] := 16#7B70;
   // GBK_TO_UNICODE[18554] := 16#B96A;
   // GBK_TO_UNICODE[18555] := 16#7B73;
   // GBK_TO_UNICODE[18556] := 16#B96B;
   // GBK_TO_UNICODE[18557] := 16#7B74;
   // GBK_TO_UNICODE[18558] := 16#B96C;
   // GBK_TO_UNICODE[18559] := 16#7B76;
   // GBK_TO_UNICODE[18560] := 16#B96D;
   // GBK_TO_UNICODE[18561] := 16#7B78;
   // GBK_TO_UNICODE[18562] := 16#B96E;
   // GBK_TO_UNICODE[18563] := 16#7B7A;
   // GBK_TO_UNICODE[18564] := 16#B96F;
   // GBK_TO_UNICODE[18565] := 16#7B7C;
   // GBK_TO_UNICODE[18566] := 16#B970;
   // GBK_TO_UNICODE[18567] := 16#7B7D;
   // GBK_TO_UNICODE[18568] := 16#B971;
   // GBK_TO_UNICODE[18569] := 16#7B7F;
   // GBK_TO_UNICODE[18570] := 16#B972;
   // GBK_TO_UNICODE[18571] := 16#7B81;
   // GBK_TO_UNICODE[18572] := 16#B973;
   // GBK_TO_UNICODE[18573] := 16#7B82;
   // GBK_TO_UNICODE[18574] := 16#B974;
   // GBK_TO_UNICODE[18575] := 16#7B83;
   // GBK_TO_UNICODE[18576] := 16#B975;
   // GBK_TO_UNICODE[18577] := 16#7B84;
   // GBK_TO_UNICODE[18578] := 16#B976;
   // GBK_TO_UNICODE[18579] := 16#7B86;
   // GBK_TO_UNICODE[18580] := 16#B977;
   // GBK_TO_UNICODE[18581] := 16#7B87;
   // GBK_TO_UNICODE[18582] := 16#B978;
   // GBK_TO_UNICODE[18583] := 16#7B88;
   // GBK_TO_UNICODE[18584] := 16#B979;
   // GBK_TO_UNICODE[18585] := 16#7B89;
   // GBK_TO_UNICODE[18586] := 16#B97A;
   // GBK_TO_UNICODE[18587] := 16#7B8A;
   // GBK_TO_UNICODE[18588] := 16#B97B;
   // GBK_TO_UNICODE[18589] := 16#7B8B;
   // GBK_TO_UNICODE[18590] := 16#B97C;
   // GBK_TO_UNICODE[18591] := 16#7B8C;
   // GBK_TO_UNICODE[18592] := 16#B97D;
   // GBK_TO_UNICODE[18593] := 16#7B8E;
   // GBK_TO_UNICODE[18594] := 16#B97E;
   // GBK_TO_UNICODE[18595] := 16#7B8F;
   // GBK_TO_UNICODE[18596] := 16#B980;
   // GBK_TO_UNICODE[18597] := 16#7B91;
   // GBK_TO_UNICODE[18598] := 16#B981;
   // GBK_TO_UNICODE[18599] := 16#7B92;
   // GBK_TO_UNICODE[18600] := 16#B982;
   // GBK_TO_UNICODE[18601] := 16#7B93;
   // GBK_TO_UNICODE[18602] := 16#B983;
   // GBK_TO_UNICODE[18603] := 16#7B96;
   // GBK_TO_UNICODE[18604] := 16#B984;
   // GBK_TO_UNICODE[18605] := 16#7B98;
   // GBK_TO_UNICODE[18606] := 16#B985;
   // GBK_TO_UNICODE[18607] := 16#7B99;
   // GBK_TO_UNICODE[18608] := 16#B986;
   // GBK_TO_UNICODE[18609] := 16#7B9A;
   // GBK_TO_UNICODE[18610] := 16#B987;
   // GBK_TO_UNICODE[18611] := 16#7B9B;
   // GBK_TO_UNICODE[18612] := 16#B988;
   // GBK_TO_UNICODE[18613] := 16#7B9E;
   // GBK_TO_UNICODE[18614] := 16#B989;
   // GBK_TO_UNICODE[18615] := 16#7B9F;
   // GBK_TO_UNICODE[18616] := 16#B98A;
   // GBK_TO_UNICODE[18617] := 16#7BA0;
   // GBK_TO_UNICODE[18618] := 16#B98B;
   // GBK_TO_UNICODE[18619] := 16#7BA3;
   // GBK_TO_UNICODE[18620] := 16#B98C;
   // GBK_TO_UNICODE[18621] := 16#7BA4;
   // GBK_TO_UNICODE[18622] := 16#B98D;
   // GBK_TO_UNICODE[18623] := 16#7BA5;
   // GBK_TO_UNICODE[18624] := 16#B98E;
   // GBK_TO_UNICODE[18625] := 16#7BAE;
   // GBK_TO_UNICODE[18626] := 16#B98F;
   // GBK_TO_UNICODE[18627] := 16#7BAF;
   // GBK_TO_UNICODE[18628] := 16#B990;
   // GBK_TO_UNICODE[18629] := 16#7BB0;
   // GBK_TO_UNICODE[18630] := 16#B991;
   // GBK_TO_UNICODE[18631] := 16#7BB2;
   // GBK_TO_UNICODE[18632] := 16#B992;
   // GBK_TO_UNICODE[18633] := 16#7BB3;
   // GBK_TO_UNICODE[18634] := 16#B993;
   // GBK_TO_UNICODE[18635] := 16#7BB5;
   // GBK_TO_UNICODE[18636] := 16#B994;
   // GBK_TO_UNICODE[18637] := 16#7BB6;
   // GBK_TO_UNICODE[18638] := 16#B995;
   // GBK_TO_UNICODE[18639] := 16#7BB7;
   // GBK_TO_UNICODE[18640] := 16#B996;
   // GBK_TO_UNICODE[18641] := 16#7BB9;
   // GBK_TO_UNICODE[18642] := 16#B997;
   // GBK_TO_UNICODE[18643] := 16#7BBA;
   // GBK_TO_UNICODE[18644] := 16#B998;
   // GBK_TO_UNICODE[18645] := 16#7BBB;
   // GBK_TO_UNICODE[18646] := 16#B999;
   // GBK_TO_UNICODE[18647] := 16#7BBC;
   // GBK_TO_UNICODE[18648] := 16#B99A;
   // GBK_TO_UNICODE[18649] := 16#7BBD;
   // GBK_TO_UNICODE[18650] := 16#B99B;
   // GBK_TO_UNICODE[18651] := 16#7BBE;
   // GBK_TO_UNICODE[18652] := 16#B99C;
   // GBK_TO_UNICODE[18653] := 16#7BBF;
   // GBK_TO_UNICODE[18654] := 16#B99D;
   // GBK_TO_UNICODE[18655] := 16#7BC0;
   // GBK_TO_UNICODE[18656] := 16#B99E;
   // GBK_TO_UNICODE[18657] := 16#7BC2;
   // GBK_TO_UNICODE[18658] := 16#B99F;
   // GBK_TO_UNICODE[18659] := 16#7BC3;
   // GBK_TO_UNICODE[18660] := 16#B9A0;
   // GBK_TO_UNICODE[18661] := 16#7BC4;
   // GBK_TO_UNICODE[18662] := 16#B9A1;
   // GBK_TO_UNICODE[18663] := 16#57C2;
   // GBK_TO_UNICODE[18664] := 16#B9A2;
   // GBK_TO_UNICODE[18665] := 16#803F;
   // GBK_TO_UNICODE[18666] := 16#B9A3;
   // GBK_TO_UNICODE[18667] := 16#6897;
   // GBK_TO_UNICODE[18668] := 16#B9A4;
   // GBK_TO_UNICODE[18669] := 16#5DE5;
   // GBK_TO_UNICODE[18670] := 16#B9A5;
   // GBK_TO_UNICODE[18671] := 16#653B;
   // GBK_TO_UNICODE[18672] := 16#B9A6;
   // GBK_TO_UNICODE[18673] := 16#529F;
   // GBK_TO_UNICODE[18674] := 16#B9A7;
   // GBK_TO_UNICODE[18675] := 16#606D;
   // GBK_TO_UNICODE[18676] := 16#B9A8;
   // GBK_TO_UNICODE[18677] := 16#9F9A;
   // GBK_TO_UNICODE[18678] := 16#B9A9;
   // GBK_TO_UNICODE[18679] := 16#4F9B;
   // GBK_TO_UNICODE[18680] := 16#B9AA;
   // GBK_TO_UNICODE[18681] := 16#8EAC;
   // GBK_TO_UNICODE[18682] := 16#B9AB;
   // GBK_TO_UNICODE[18683] := 16#516C;
   // GBK_TO_UNICODE[18684] := 16#B9AC;
   // GBK_TO_UNICODE[18685] := 16#5BAB;
   // GBK_TO_UNICODE[18686] := 16#B9AD;
   // GBK_TO_UNICODE[18687] := 16#5F13;
   // GBK_TO_UNICODE[18688] := 16#B9AE;
   // GBK_TO_UNICODE[18689] := 16#5DE9;
   // GBK_TO_UNICODE[18690] := 16#B9AF;
   // GBK_TO_UNICODE[18691] := 16#6C5E;
   // GBK_TO_UNICODE[18692] := 16#B9B0;
   // GBK_TO_UNICODE[18693] := 16#62F1;
   // GBK_TO_UNICODE[18694] := 16#B9B1;
   // GBK_TO_UNICODE[18695] := 16#8D21;
   // GBK_TO_UNICODE[18696] := 16#B9B2;
   // GBK_TO_UNICODE[18697] := 16#5171;
   // GBK_TO_UNICODE[18698] := 16#B9B3;
   // GBK_TO_UNICODE[18699] := 16#94A9;
   // GBK_TO_UNICODE[18700] := 16#B9B4;
   // GBK_TO_UNICODE[18701] := 16#52FE;
   // GBK_TO_UNICODE[18702] := 16#B9B5;
   // GBK_TO_UNICODE[18703] := 16#6C9F;
   // GBK_TO_UNICODE[18704] := 16#B9B6;
   // GBK_TO_UNICODE[18705] := 16#82DF;
   // GBK_TO_UNICODE[18706] := 16#B9B7;
   // GBK_TO_UNICODE[18707] := 16#72D7;
   // GBK_TO_UNICODE[18708] := 16#B9B8;
   // GBK_TO_UNICODE[18709] := 16#57A2;
   // GBK_TO_UNICODE[18710] := 16#B9B9;
   // GBK_TO_UNICODE[18711] := 16#6784;
   // GBK_TO_UNICODE[18712] := 16#B9BA;
   // GBK_TO_UNICODE[18713] := 16#8D2D;
   // GBK_TO_UNICODE[18714] := 16#B9BB;
   // GBK_TO_UNICODE[18715] := 16#591F;
   // GBK_TO_UNICODE[18716] := 16#B9BC;
   // GBK_TO_UNICODE[18717] := 16#8F9C;
   // GBK_TO_UNICODE[18718] := 16#B9BD;
   // GBK_TO_UNICODE[18719] := 16#83C7;
   // GBK_TO_UNICODE[18720] := 16#B9BE;
   // GBK_TO_UNICODE[18721] := 16#5495;
   // GBK_TO_UNICODE[18722] := 16#B9BF;
   // GBK_TO_UNICODE[18723] := 16#7B8D;
   // GBK_TO_UNICODE[18724] := 16#B9C0;
   // GBK_TO_UNICODE[18725] := 16#4F30;
   // GBK_TO_UNICODE[18726] := 16#B9C1;
   // GBK_TO_UNICODE[18727] := 16#6CBD;
   // GBK_TO_UNICODE[18728] := 16#B9C2;
   // GBK_TO_UNICODE[18729] := 16#5B64;
   // GBK_TO_UNICODE[18730] := 16#B9C3;
   // GBK_TO_UNICODE[18731] := 16#59D1;
   // GBK_TO_UNICODE[18732] := 16#B9C4;
   // GBK_TO_UNICODE[18733] := 16#9F13;
   // GBK_TO_UNICODE[18734] := 16#B9C5;
   // GBK_TO_UNICODE[18735] := 16#53E4;
   // GBK_TO_UNICODE[18736] := 16#B9C6;
   // GBK_TO_UNICODE[18737] := 16#86CA;
   // GBK_TO_UNICODE[18738] := 16#B9C7;
   // GBK_TO_UNICODE[18739] := 16#9AA8;
   // GBK_TO_UNICODE[18740] := 16#B9C8;
   // GBK_TO_UNICODE[18741] := 16#8C37;
   // GBK_TO_UNICODE[18742] := 16#B9C9;
   // GBK_TO_UNICODE[18743] := 16#80A1;
   // GBK_TO_UNICODE[18744] := 16#B9CA;
   // GBK_TO_UNICODE[18745] := 16#6545;
   // GBK_TO_UNICODE[18746] := 16#B9CB;
   // GBK_TO_UNICODE[18747] := 16#987E;
   // GBK_TO_UNICODE[18748] := 16#B9CC;
   // GBK_TO_UNICODE[18749] := 16#56FA;
   // GBK_TO_UNICODE[18750] := 16#B9CD;
   // GBK_TO_UNICODE[18751] := 16#96C7;
   // GBK_TO_UNICODE[18752] := 16#B9CE;
   // GBK_TO_UNICODE[18753] := 16#522E;
   // GBK_TO_UNICODE[18754] := 16#B9CF;
   // GBK_TO_UNICODE[18755] := 16#74DC;
   // GBK_TO_UNICODE[18756] := 16#B9D0;
   // GBK_TO_UNICODE[18757] := 16#5250;
   // GBK_TO_UNICODE[18758] := 16#B9D1;
   // GBK_TO_UNICODE[18759] := 16#5BE1;
   // GBK_TO_UNICODE[18760] := 16#B9D2;
   // GBK_TO_UNICODE[18761] := 16#6302;
   // GBK_TO_UNICODE[18762] := 16#B9D3;
   // GBK_TO_UNICODE[18763] := 16#8902;
   // GBK_TO_UNICODE[18764] := 16#B9D4;
   // GBK_TO_UNICODE[18765] := 16#4E56;
   // GBK_TO_UNICODE[18766] := 16#B9D5;
   // GBK_TO_UNICODE[18767] := 16#62D0;
   // GBK_TO_UNICODE[18768] := 16#B9D6;
   // GBK_TO_UNICODE[18769] := 16#602A;
   // GBK_TO_UNICODE[18770] := 16#B9D7;
   // GBK_TO_UNICODE[18771] := 16#68FA;
   // GBK_TO_UNICODE[18772] := 16#B9D8;
   // GBK_TO_UNICODE[18773] := 16#5173;
   // GBK_TO_UNICODE[18774] := 16#B9D9;
   // GBK_TO_UNICODE[18775] := 16#5B98;
   // GBK_TO_UNICODE[18776] := 16#B9DA;
   // GBK_TO_UNICODE[18777] := 16#51A0;
   // GBK_TO_UNICODE[18778] := 16#B9DB;
   // GBK_TO_UNICODE[18779] := 16#89C2;
   // GBK_TO_UNICODE[18780] := 16#B9DC;
   // GBK_TO_UNICODE[18781] := 16#7BA1;
   // GBK_TO_UNICODE[18782] := 16#B9DD;
   // GBK_TO_UNICODE[18783] := 16#9986;
   // GBK_TO_UNICODE[18784] := 16#B9DE;
   // GBK_TO_UNICODE[18785] := 16#7F50;
   // GBK_TO_UNICODE[18786] := 16#B9DF;
   // GBK_TO_UNICODE[18787] := 16#60EF;
   // GBK_TO_UNICODE[18788] := 16#B9E0;
   // GBK_TO_UNICODE[18789] := 16#704C;
   // GBK_TO_UNICODE[18790] := 16#B9E1;
   // GBK_TO_UNICODE[18791] := 16#8D2F;
   // GBK_TO_UNICODE[18792] := 16#B9E2;
   // GBK_TO_UNICODE[18793] := 16#5149;
   // GBK_TO_UNICODE[18794] := 16#B9E3;
   // GBK_TO_UNICODE[18795] := 16#5E7F;
   // GBK_TO_UNICODE[18796] := 16#B9E4;
   // GBK_TO_UNICODE[18797] := 16#901B;
   // GBK_TO_UNICODE[18798] := 16#B9E5;
   // GBK_TO_UNICODE[18799] := 16#7470;
   // GBK_TO_UNICODE[18800] := 16#B9E6;
   // GBK_TO_UNICODE[18801] := 16#89C4;
   // GBK_TO_UNICODE[18802] := 16#B9E7;
   // GBK_TO_UNICODE[18803] := 16#572D;
   // GBK_TO_UNICODE[18804] := 16#B9E8;
   // GBK_TO_UNICODE[18805] := 16#7845;
   // GBK_TO_UNICODE[18806] := 16#B9E9;
   // GBK_TO_UNICODE[18807] := 16#5F52;
   // GBK_TO_UNICODE[18808] := 16#B9EA;
   // GBK_TO_UNICODE[18809] := 16#9F9F;
   // GBK_TO_UNICODE[18810] := 16#B9EB;
   // GBK_TO_UNICODE[18811] := 16#95FA;
   // GBK_TO_UNICODE[18812] := 16#B9EC;
   // GBK_TO_UNICODE[18813] := 16#8F68;
   // GBK_TO_UNICODE[18814] := 16#B9ED;
   // GBK_TO_UNICODE[18815] := 16#9B3C;
   // GBK_TO_UNICODE[18816] := 16#B9EE;
   // GBK_TO_UNICODE[18817] := 16#8BE1;
   // GBK_TO_UNICODE[18818] := 16#B9EF;
   // GBK_TO_UNICODE[18819] := 16#7678;
   // GBK_TO_UNICODE[18820] := 16#B9F0;
   // GBK_TO_UNICODE[18821] := 16#6842;
   // GBK_TO_UNICODE[18822] := 16#B9F1;
   // GBK_TO_UNICODE[18823] := 16#67DC;
   // GBK_TO_UNICODE[18824] := 16#B9F2;
   // GBK_TO_UNICODE[18825] := 16#8DEA;
   // GBK_TO_UNICODE[18826] := 16#B9F3;
   // GBK_TO_UNICODE[18827] := 16#8D35;
   // GBK_TO_UNICODE[18828] := 16#B9F4;
   // GBK_TO_UNICODE[18829] := 16#523D;
   // GBK_TO_UNICODE[18830] := 16#B9F5;
   // GBK_TO_UNICODE[18831] := 16#8F8A;
   // GBK_TO_UNICODE[18832] := 16#B9F6;
   // GBK_TO_UNICODE[18833] := 16#6EDA;
   // GBK_TO_UNICODE[18834] := 16#B9F7;
   // GBK_TO_UNICODE[18835] := 16#68CD;
   // GBK_TO_UNICODE[18836] := 16#B9F8;
   // GBK_TO_UNICODE[18837] := 16#9505;
   // GBK_TO_UNICODE[18838] := 16#B9F9;
   // GBK_TO_UNICODE[18839] := 16#90ED;
   // GBK_TO_UNICODE[18840] := 16#B9FA;
   // GBK_TO_UNICODE[18841] := 16#56FD;
   // GBK_TO_UNICODE[18842] := 16#B9FB;
   // GBK_TO_UNICODE[18843] := 16#679C;
   // GBK_TO_UNICODE[18844] := 16#B9FC;
   // GBK_TO_UNICODE[18845] := 16#88F9;
   // GBK_TO_UNICODE[18846] := 16#B9FD;
   // GBK_TO_UNICODE[18847] := 16#8FC7;
   // GBK_TO_UNICODE[18848] := 16#B9FE;
   // GBK_TO_UNICODE[18849] := 16#54C8;
   // GBK_TO_UNICODE[18850] := 16#BA40;
   // GBK_TO_UNICODE[18851] := 16#7BC5;
   // GBK_TO_UNICODE[18852] := 16#BA41;
   // GBK_TO_UNICODE[18853] := 16#7BC8;
   // GBK_TO_UNICODE[18854] := 16#BA42;
   // GBK_TO_UNICODE[18855] := 16#7BC9;
   // GBK_TO_UNICODE[18856] := 16#BA43;
   // GBK_TO_UNICODE[18857] := 16#7BCA;
   // GBK_TO_UNICODE[18858] := 16#BA44;
   // GBK_TO_UNICODE[18859] := 16#7BCB;
   // GBK_TO_UNICODE[18860] := 16#BA45;
   // GBK_TO_UNICODE[18861] := 16#7BCD;
   // GBK_TO_UNICODE[18862] := 16#BA46;
   // GBK_TO_UNICODE[18863] := 16#7BCE;
   // GBK_TO_UNICODE[18864] := 16#BA47;
   // GBK_TO_UNICODE[18865] := 16#7BCF;
   // GBK_TO_UNICODE[18866] := 16#BA48;
   // GBK_TO_UNICODE[18867] := 16#7BD0;
   // GBK_TO_UNICODE[18868] := 16#BA49;
   // GBK_TO_UNICODE[18869] := 16#7BD2;
   // GBK_TO_UNICODE[18870] := 16#BA4A;
   // GBK_TO_UNICODE[18871] := 16#7BD4;
   // GBK_TO_UNICODE[18872] := 16#BA4B;
   // GBK_TO_UNICODE[18873] := 16#7BD5;
   // GBK_TO_UNICODE[18874] := 16#BA4C;
   // GBK_TO_UNICODE[18875] := 16#7BD6;
   // GBK_TO_UNICODE[18876] := 16#BA4D;
   // GBK_TO_UNICODE[18877] := 16#7BD7;
   // GBK_TO_UNICODE[18878] := 16#BA4E;
   // GBK_TO_UNICODE[18879] := 16#7BD8;
   // GBK_TO_UNICODE[18880] := 16#BA4F;
   // GBK_TO_UNICODE[18881] := 16#7BDB;
   // GBK_TO_UNICODE[18882] := 16#BA50;
   // GBK_TO_UNICODE[18883] := 16#7BDC;
   // GBK_TO_UNICODE[18884] := 16#BA51;
   // GBK_TO_UNICODE[18885] := 16#7BDE;
   // GBK_TO_UNICODE[18886] := 16#BA52;
   // GBK_TO_UNICODE[18887] := 16#7BDF;
   // GBK_TO_UNICODE[18888] := 16#BA53;
   // GBK_TO_UNICODE[18889] := 16#7BE0;
   // GBK_TO_UNICODE[18890] := 16#BA54;
   // GBK_TO_UNICODE[18891] := 16#7BE2;
   // GBK_TO_UNICODE[18892] := 16#BA55;
   // GBK_TO_UNICODE[18893] := 16#7BE3;
   // GBK_TO_UNICODE[18894] := 16#BA56;
   // GBK_TO_UNICODE[18895] := 16#7BE4;
   // GBK_TO_UNICODE[18896] := 16#BA57;
   // GBK_TO_UNICODE[18897] := 16#7BE7;
   // GBK_TO_UNICODE[18898] := 16#BA58;
   // GBK_TO_UNICODE[18899] := 16#7BE8;
   // GBK_TO_UNICODE[18900] := 16#BA59;
   // GBK_TO_UNICODE[18901] := 16#7BE9;
   // GBK_TO_UNICODE[18902] := 16#BA5A;
   // GBK_TO_UNICODE[18903] := 16#7BEB;
   // GBK_TO_UNICODE[18904] := 16#BA5B;
   // GBK_TO_UNICODE[18905] := 16#7BEC;
   // GBK_TO_UNICODE[18906] := 16#BA5C;
   // GBK_TO_UNICODE[18907] := 16#7BED;
   // GBK_TO_UNICODE[18908] := 16#BA5D;
   // GBK_TO_UNICODE[18909] := 16#7BEF;
   // GBK_TO_UNICODE[18910] := 16#BA5E;
   // GBK_TO_UNICODE[18911] := 16#7BF0;
   // GBK_TO_UNICODE[18912] := 16#BA5F;
   // GBK_TO_UNICODE[18913] := 16#7BF2;
   // GBK_TO_UNICODE[18914] := 16#BA60;
   // GBK_TO_UNICODE[18915] := 16#7BF3;
   // GBK_TO_UNICODE[18916] := 16#BA61;
   // GBK_TO_UNICODE[18917] := 16#7BF4;
   // GBK_TO_UNICODE[18918] := 16#BA62;
   // GBK_TO_UNICODE[18919] := 16#7BF5;
   // GBK_TO_UNICODE[18920] := 16#BA63;
   // GBK_TO_UNICODE[18921] := 16#7BF6;
   // GBK_TO_UNICODE[18922] := 16#BA64;
   // GBK_TO_UNICODE[18923] := 16#7BF8;
   // GBK_TO_UNICODE[18924] := 16#BA65;
   // GBK_TO_UNICODE[18925] := 16#7BF9;
   // GBK_TO_UNICODE[18926] := 16#BA66;
   // GBK_TO_UNICODE[18927] := 16#7BFA;
   // GBK_TO_UNICODE[18928] := 16#BA67;
   // GBK_TO_UNICODE[18929] := 16#7BFB;
   // GBK_TO_UNICODE[18930] := 16#BA68;
   // GBK_TO_UNICODE[18931] := 16#7BFD;
   // GBK_TO_UNICODE[18932] := 16#BA69;
   // GBK_TO_UNICODE[18933] := 16#7BFF;
   // GBK_TO_UNICODE[18934] := 16#BA6A;
   // GBK_TO_UNICODE[18935] := 16#7C00;
   // GBK_TO_UNICODE[18936] := 16#BA6B;
   // GBK_TO_UNICODE[18937] := 16#7C01;
   // GBK_TO_UNICODE[18938] := 16#BA6C;
   // GBK_TO_UNICODE[18939] := 16#7C02;
   // GBK_TO_UNICODE[18940] := 16#BA6D;
   // GBK_TO_UNICODE[18941] := 16#7C03;
   // GBK_TO_UNICODE[18942] := 16#BA6E;
   // GBK_TO_UNICODE[18943] := 16#7C04;
   // GBK_TO_UNICODE[18944] := 16#BA6F;
   // GBK_TO_UNICODE[18945] := 16#7C05;
   // GBK_TO_UNICODE[18946] := 16#BA70;
   // GBK_TO_UNICODE[18947] := 16#7C06;
   // GBK_TO_UNICODE[18948] := 16#BA71;
   // GBK_TO_UNICODE[18949] := 16#7C08;
   // GBK_TO_UNICODE[18950] := 16#BA72;
   // GBK_TO_UNICODE[18951] := 16#7C09;
   // GBK_TO_UNICODE[18952] := 16#BA73;
   // GBK_TO_UNICODE[18953] := 16#7C0A;
   // GBK_TO_UNICODE[18954] := 16#BA74;
   // GBK_TO_UNICODE[18955] := 16#7C0D;
   // GBK_TO_UNICODE[18956] := 16#BA75;
   // GBK_TO_UNICODE[18957] := 16#7C0E;
   // GBK_TO_UNICODE[18958] := 16#BA76;
   // GBK_TO_UNICODE[18959] := 16#7C10;
   // GBK_TO_UNICODE[18960] := 16#BA77;
   // GBK_TO_UNICODE[18961] := 16#7C11;
   // GBK_TO_UNICODE[18962] := 16#BA78;
   // GBK_TO_UNICODE[18963] := 16#7C12;
   // GBK_TO_UNICODE[18964] := 16#BA79;
   // GBK_TO_UNICODE[18965] := 16#7C13;
   // GBK_TO_UNICODE[18966] := 16#BA7A;
   // GBK_TO_UNICODE[18967] := 16#7C14;
   // GBK_TO_UNICODE[18968] := 16#BA7B;
   // GBK_TO_UNICODE[18969] := 16#7C15;
   // GBK_TO_UNICODE[18970] := 16#BA7C;
   // GBK_TO_UNICODE[18971] := 16#7C17;
   // GBK_TO_UNICODE[18972] := 16#BA7D;
   // GBK_TO_UNICODE[18973] := 16#7C18;
   // GBK_TO_UNICODE[18974] := 16#BA7E;
   // GBK_TO_UNICODE[18975] := 16#7C19;
   // GBK_TO_UNICODE[18976] := 16#BA80;
   // GBK_TO_UNICODE[18977] := 16#7C1A;
   // GBK_TO_UNICODE[18978] := 16#BA81;
   // GBK_TO_UNICODE[18979] := 16#7C1B;
   // GBK_TO_UNICODE[18980] := 16#BA82;
   // GBK_TO_UNICODE[18981] := 16#7C1C;
   // GBK_TO_UNICODE[18982] := 16#BA83;
   // GBK_TO_UNICODE[18983] := 16#7C1D;
   // GBK_TO_UNICODE[18984] := 16#BA84;
   // GBK_TO_UNICODE[18985] := 16#7C1E;
   // GBK_TO_UNICODE[18986] := 16#BA85;
   // GBK_TO_UNICODE[18987] := 16#7C20;
   // GBK_TO_UNICODE[18988] := 16#BA86;
   // GBK_TO_UNICODE[18989] := 16#7C21;
   // GBK_TO_UNICODE[18990] := 16#BA87;
   // GBK_TO_UNICODE[18991] := 16#7C22;
   // GBK_TO_UNICODE[18992] := 16#BA88;
   // GBK_TO_UNICODE[18993] := 16#7C23;
   // GBK_TO_UNICODE[18994] := 16#BA89;
   // GBK_TO_UNICODE[18995] := 16#7C24;
   // GBK_TO_UNICODE[18996] := 16#BA8A;
   // GBK_TO_UNICODE[18997] := 16#7C25;
   // GBK_TO_UNICODE[18998] := 16#BA8B;
   // GBK_TO_UNICODE[18999] := 16#7C28;
   // GBK_TO_UNICODE[19000] := 16#BA8C;
   // GBK_TO_UNICODE[19001] := 16#7C29;
   // GBK_TO_UNICODE[19002] := 16#BA8D;
   // GBK_TO_UNICODE[19003] := 16#7C2B;
   // GBK_TO_UNICODE[19004] := 16#BA8E;
   // GBK_TO_UNICODE[19005] := 16#7C2C;
   // GBK_TO_UNICODE[19006] := 16#BA8F;
   // GBK_TO_UNICODE[19007] := 16#7C2D;
   // GBK_TO_UNICODE[19008] := 16#BA90;
   // GBK_TO_UNICODE[19009] := 16#7C2E;
   // GBK_TO_UNICODE[19010] := 16#BA91;
   // GBK_TO_UNICODE[19011] := 16#7C2F;
   // GBK_TO_UNICODE[19012] := 16#BA92;
   // GBK_TO_UNICODE[19013] := 16#7C30;
   // GBK_TO_UNICODE[19014] := 16#BA93;
   // GBK_TO_UNICODE[19015] := 16#7C31;
   // GBK_TO_UNICODE[19016] := 16#BA94;
   // GBK_TO_UNICODE[19017] := 16#7C32;
   // GBK_TO_UNICODE[19018] := 16#BA95;
   // GBK_TO_UNICODE[19019] := 16#7C33;
   // GBK_TO_UNICODE[19020] := 16#BA96;
   // GBK_TO_UNICODE[19021] := 16#7C34;
   // GBK_TO_UNICODE[19022] := 16#BA97;
   // GBK_TO_UNICODE[19023] := 16#7C35;
   // GBK_TO_UNICODE[19024] := 16#BA98;
   // GBK_TO_UNICODE[19025] := 16#7C36;
   // GBK_TO_UNICODE[19026] := 16#BA99;
   // GBK_TO_UNICODE[19027] := 16#7C37;
   // GBK_TO_UNICODE[19028] := 16#BA9A;
   // GBK_TO_UNICODE[19029] := 16#7C39;
   // GBK_TO_UNICODE[19030] := 16#BA9B;
   // GBK_TO_UNICODE[19031] := 16#7C3A;
   // GBK_TO_UNICODE[19032] := 16#BA9C;
   // GBK_TO_UNICODE[19033] := 16#7C3B;
   // GBK_TO_UNICODE[19034] := 16#BA9D;
   // GBK_TO_UNICODE[19035] := 16#7C3C;
   // GBK_TO_UNICODE[19036] := 16#BA9E;
   // GBK_TO_UNICODE[19037] := 16#7C3D;
   // GBK_TO_UNICODE[19038] := 16#BA9F;
   // GBK_TO_UNICODE[19039] := 16#7C3E;
   // GBK_TO_UNICODE[19040] := 16#BAA0;
   // GBK_TO_UNICODE[19041] := 16#7C42;
   // GBK_TO_UNICODE[19042] := 16#BAA1;
   // GBK_TO_UNICODE[19043] := 16#9AB8;
   // GBK_TO_UNICODE[19044] := 16#BAA2;
   // GBK_TO_UNICODE[19045] := 16#5B69;
   // GBK_TO_UNICODE[19046] := 16#BAA3;
   // GBK_TO_UNICODE[19047] := 16#6D77;
   // GBK_TO_UNICODE[19048] := 16#BAA4;
   // GBK_TO_UNICODE[19049] := 16#6C26;
   // GBK_TO_UNICODE[19050] := 16#BAA5;
   // GBK_TO_UNICODE[19051] := 16#4EA5;
   // GBK_TO_UNICODE[19052] := 16#BAA6;
   // GBK_TO_UNICODE[19053] := 16#5BB3;
   // GBK_TO_UNICODE[19054] := 16#BAA7;
   // GBK_TO_UNICODE[19055] := 16#9A87;
   // GBK_TO_UNICODE[19056] := 16#BAA8;
   // GBK_TO_UNICODE[19057] := 16#9163;
   // GBK_TO_UNICODE[19058] := 16#BAA9;
   // GBK_TO_UNICODE[19059] := 16#61A8;
   // GBK_TO_UNICODE[19060] := 16#BAAA;
   // GBK_TO_UNICODE[19061] := 16#90AF;
   // GBK_TO_UNICODE[19062] := 16#BAAB;
   // GBK_TO_UNICODE[19063] := 16#97E9;
   // GBK_TO_UNICODE[19064] := 16#BAAC;
   // GBK_TO_UNICODE[19065] := 16#542B;
   // GBK_TO_UNICODE[19066] := 16#BAAD;
   // GBK_TO_UNICODE[19067] := 16#6DB5;
   // GBK_TO_UNICODE[19068] := 16#BAAE;
   // GBK_TO_UNICODE[19069] := 16#5BD2;
   // GBK_TO_UNICODE[19070] := 16#BAAF;
   // GBK_TO_UNICODE[19071] := 16#51FD;
   // GBK_TO_UNICODE[19072] := 16#BAB0;
   // GBK_TO_UNICODE[19073] := 16#558A;
   // GBK_TO_UNICODE[19074] := 16#BAB1;
   // GBK_TO_UNICODE[19075] := 16#7F55;
   // GBK_TO_UNICODE[19076] := 16#BAB2;
   // GBK_TO_UNICODE[19077] := 16#7FF0;
   // GBK_TO_UNICODE[19078] := 16#BAB3;
   // GBK_TO_UNICODE[19079] := 16#64BC;
   // GBK_TO_UNICODE[19080] := 16#BAB4;
   // GBK_TO_UNICODE[19081] := 16#634D;
   // GBK_TO_UNICODE[19082] := 16#BAB5;
   // GBK_TO_UNICODE[19083] := 16#65F1;
   // GBK_TO_UNICODE[19084] := 16#BAB6;
   // GBK_TO_UNICODE[19085] := 16#61BE;
   // GBK_TO_UNICODE[19086] := 16#BAB7;
   // GBK_TO_UNICODE[19087] := 16#608D;
   // GBK_TO_UNICODE[19088] := 16#BAB8;
   // GBK_TO_UNICODE[19089] := 16#710A;
   // GBK_TO_UNICODE[19090] := 16#BAB9;
   // GBK_TO_UNICODE[19091] := 16#6C57;
   // GBK_TO_UNICODE[19092] := 16#BABA;
   // GBK_TO_UNICODE[19093] := 16#6C49;
   // GBK_TO_UNICODE[19094] := 16#BABB;
   // GBK_TO_UNICODE[19095] := 16#592F;
   // GBK_TO_UNICODE[19096] := 16#BABC;
   // GBK_TO_UNICODE[19097] := 16#676D;
   // GBK_TO_UNICODE[19098] := 16#BABD;
   // GBK_TO_UNICODE[19099] := 16#822A;
   // GBK_TO_UNICODE[19100] := 16#BABE;
   // GBK_TO_UNICODE[19101] := 16#58D5;
   // GBK_TO_UNICODE[19102] := 16#BABF;
   // GBK_TO_UNICODE[19103] := 16#568E;
   // GBK_TO_UNICODE[19104] := 16#BAC0;
   // GBK_TO_UNICODE[19105] := 16#8C6A;
   // GBK_TO_UNICODE[19106] := 16#BAC1;
   // GBK_TO_UNICODE[19107] := 16#6BEB;
   // GBK_TO_UNICODE[19108] := 16#BAC2;
   // GBK_TO_UNICODE[19109] := 16#90DD;
   // GBK_TO_UNICODE[19110] := 16#BAC3;
   // GBK_TO_UNICODE[19111] := 16#597D;
   // GBK_TO_UNICODE[19112] := 16#BAC4;
   // GBK_TO_UNICODE[19113] := 16#8017;
   // GBK_TO_UNICODE[19114] := 16#BAC5;
   // GBK_TO_UNICODE[19115] := 16#53F7;
   // GBK_TO_UNICODE[19116] := 16#BAC6;
   // GBK_TO_UNICODE[19117] := 16#6D69;
   // GBK_TO_UNICODE[19118] := 16#BAC7;
   // GBK_TO_UNICODE[19119] := 16#5475;
   // GBK_TO_UNICODE[19120] := 16#BAC8;
   // GBK_TO_UNICODE[19121] := 16#559D;
   // GBK_TO_UNICODE[19122] := 16#BAC9;
   // GBK_TO_UNICODE[19123] := 16#8377;
   // GBK_TO_UNICODE[19124] := 16#BACA;
   // GBK_TO_UNICODE[19125] := 16#83CF;
   // GBK_TO_UNICODE[19126] := 16#BACB;
   // GBK_TO_UNICODE[19127] := 16#6838;
   // GBK_TO_UNICODE[19128] := 16#BACC;
   // GBK_TO_UNICODE[19129] := 16#79BE;
   // GBK_TO_UNICODE[19130] := 16#BACD;
   // GBK_TO_UNICODE[19131] := 16#548C;
   // GBK_TO_UNICODE[19132] := 16#BACE;
   // GBK_TO_UNICODE[19133] := 16#4F55;
   // GBK_TO_UNICODE[19134] := 16#BACF;
   // GBK_TO_UNICODE[19135] := 16#5408;
   // GBK_TO_UNICODE[19136] := 16#BAD0;
   // GBK_TO_UNICODE[19137] := 16#76D2;
   // GBK_TO_UNICODE[19138] := 16#BAD1;
   // GBK_TO_UNICODE[19139] := 16#8C89;
   // GBK_TO_UNICODE[19140] := 16#BAD2;
   // GBK_TO_UNICODE[19141] := 16#9602;
   // GBK_TO_UNICODE[19142] := 16#BAD3;
   // GBK_TO_UNICODE[19143] := 16#6CB3;
   // GBK_TO_UNICODE[19144] := 16#BAD4;
   // GBK_TO_UNICODE[19145] := 16#6DB8;
   // GBK_TO_UNICODE[19146] := 16#BAD5;
   // GBK_TO_UNICODE[19147] := 16#8D6B;
   // GBK_TO_UNICODE[19148] := 16#BAD6;
   // GBK_TO_UNICODE[19149] := 16#8910;
   // GBK_TO_UNICODE[19150] := 16#BAD7;
   // GBK_TO_UNICODE[19151] := 16#9E64;
   // GBK_TO_UNICODE[19152] := 16#BAD8;
   // GBK_TO_UNICODE[19153] := 16#8D3A;
   // GBK_TO_UNICODE[19154] := 16#BAD9;
   // GBK_TO_UNICODE[19155] := 16#563F;
   // GBK_TO_UNICODE[19156] := 16#BADA;
   // GBK_TO_UNICODE[19157] := 16#9ED1;
   // GBK_TO_UNICODE[19158] := 16#BADB;
   // GBK_TO_UNICODE[19159] := 16#75D5;
   // GBK_TO_UNICODE[19160] := 16#BADC;
   // GBK_TO_UNICODE[19161] := 16#5F88;
   // GBK_TO_UNICODE[19162] := 16#BADD;
   // GBK_TO_UNICODE[19163] := 16#72E0;
   // GBK_TO_UNICODE[19164] := 16#BADE;
   // GBK_TO_UNICODE[19165] := 16#6068;
   // GBK_TO_UNICODE[19166] := 16#BADF;
   // GBK_TO_UNICODE[19167] := 16#54FC;
   // GBK_TO_UNICODE[19168] := 16#BAE0;
   // GBK_TO_UNICODE[19169] := 16#4EA8;
   // GBK_TO_UNICODE[19170] := 16#BAE1;
   // GBK_TO_UNICODE[19171] := 16#6A2A;
   // GBK_TO_UNICODE[19172] := 16#BAE2;
   // GBK_TO_UNICODE[19173] := 16#8861;
   // GBK_TO_UNICODE[19174] := 16#BAE3;
   // GBK_TO_UNICODE[19175] := 16#6052;
   // GBK_TO_UNICODE[19176] := 16#BAE4;
   // GBK_TO_UNICODE[19177] := 16#8F70;
   // GBK_TO_UNICODE[19178] := 16#BAE5;
   // GBK_TO_UNICODE[19179] := 16#54C4;
   // GBK_TO_UNICODE[19180] := 16#BAE6;
   // GBK_TO_UNICODE[19181] := 16#70D8;
   // GBK_TO_UNICODE[19182] := 16#BAE7;
   // GBK_TO_UNICODE[19183] := 16#8679;
   // GBK_TO_UNICODE[19184] := 16#BAE8;
   // GBK_TO_UNICODE[19185] := 16#9E3F;
   // GBK_TO_UNICODE[19186] := 16#BAE9;
   // GBK_TO_UNICODE[19187] := 16#6D2A;
   // GBK_TO_UNICODE[19188] := 16#BAEA;
   // GBK_TO_UNICODE[19189] := 16#5B8F;
   // GBK_TO_UNICODE[19190] := 16#BAEB;
   // GBK_TO_UNICODE[19191] := 16#5F18;
   // GBK_TO_UNICODE[19192] := 16#BAEC;
   // GBK_TO_UNICODE[19193] := 16#7EA2;
   // GBK_TO_UNICODE[19194] := 16#BAED;
   // GBK_TO_UNICODE[19195] := 16#5589;
   // GBK_TO_UNICODE[19196] := 16#BAEE;
   // GBK_TO_UNICODE[19197] := 16#4FAF;
   // GBK_TO_UNICODE[19198] := 16#BAEF;
   // GBK_TO_UNICODE[19199] := 16#7334;
   // GBK_TO_UNICODE[19200] := 16#BAF0;
   // GBK_TO_UNICODE[19201] := 16#543C;
   // GBK_TO_UNICODE[19202] := 16#BAF1;
   // GBK_TO_UNICODE[19203] := 16#539A;
   // GBK_TO_UNICODE[19204] := 16#BAF2;
   // GBK_TO_UNICODE[19205] := 16#5019;
   // GBK_TO_UNICODE[19206] := 16#BAF3;
   // GBK_TO_UNICODE[19207] := 16#540E;
   // GBK_TO_UNICODE[19208] := 16#BAF4;
   // GBK_TO_UNICODE[19209] := 16#547C;
   // GBK_TO_UNICODE[19210] := 16#BAF5;
   // GBK_TO_UNICODE[19211] := 16#4E4E;
   // GBK_TO_UNICODE[19212] := 16#BAF6;
   // GBK_TO_UNICODE[19213] := 16#5FFD;
   // GBK_TO_UNICODE[19214] := 16#BAF7;
   // GBK_TO_UNICODE[19215] := 16#745A;
   // GBK_TO_UNICODE[19216] := 16#BAF8;
   // GBK_TO_UNICODE[19217] := 16#58F6;
   // GBK_TO_UNICODE[19218] := 16#BAF9;
   // GBK_TO_UNICODE[19219] := 16#846B;
   // GBK_TO_UNICODE[19220] := 16#BAFA;
   // GBK_TO_UNICODE[19221] := 16#80E1;
   // GBK_TO_UNICODE[19222] := 16#BAFB;
   // GBK_TO_UNICODE[19223] := 16#8774;
   // GBK_TO_UNICODE[19224] := 16#BAFC;
   // GBK_TO_UNICODE[19225] := 16#72D0;
   // GBK_TO_UNICODE[19226] := 16#BAFD;
   // GBK_TO_UNICODE[19227] := 16#7CCA;
   // GBK_TO_UNICODE[19228] := 16#BAFE;
   // GBK_TO_UNICODE[19229] := 16#6E56;
   // GBK_TO_UNICODE[19230] := 16#BB40;
   // GBK_TO_UNICODE[19231] := 16#7C43;
   // GBK_TO_UNICODE[19232] := 16#BB41;
   // GBK_TO_UNICODE[19233] := 16#7C44;
   // GBK_TO_UNICODE[19234] := 16#BB42;
   // GBK_TO_UNICODE[19235] := 16#7C45;
   // GBK_TO_UNICODE[19236] := 16#BB43;
   // GBK_TO_UNICODE[19237] := 16#7C46;
   // GBK_TO_UNICODE[19238] := 16#BB44;
   // GBK_TO_UNICODE[19239] := 16#7C47;
   // GBK_TO_UNICODE[19240] := 16#BB45;
   // GBK_TO_UNICODE[19241] := 16#7C48;
   // GBK_TO_UNICODE[19242] := 16#BB46;
   // GBK_TO_UNICODE[19243] := 16#7C49;
   // GBK_TO_UNICODE[19244] := 16#BB47;
   // GBK_TO_UNICODE[19245] := 16#7C4A;
   // GBK_TO_UNICODE[19246] := 16#BB48;
   // GBK_TO_UNICODE[19247] := 16#7C4B;
   // GBK_TO_UNICODE[19248] := 16#BB49;
   // GBK_TO_UNICODE[19249] := 16#7C4C;
   // GBK_TO_UNICODE[19250] := 16#BB4A;
   // GBK_TO_UNICODE[19251] := 16#7C4E;
   // GBK_TO_UNICODE[19252] := 16#BB4B;
   // GBK_TO_UNICODE[19253] := 16#7C4F;
   // GBK_TO_UNICODE[19254] := 16#BB4C;
   // GBK_TO_UNICODE[19255] := 16#7C50;
   // GBK_TO_UNICODE[19256] := 16#BB4D;
   // GBK_TO_UNICODE[19257] := 16#7C51;
   // GBK_TO_UNICODE[19258] := 16#BB4E;
   // GBK_TO_UNICODE[19259] := 16#7C52;
   // GBK_TO_UNICODE[19260] := 16#BB4F;
   // GBK_TO_UNICODE[19261] := 16#7C53;
   // GBK_TO_UNICODE[19262] := 16#BB50;
   // GBK_TO_UNICODE[19263] := 16#7C54;
   // GBK_TO_UNICODE[19264] := 16#BB51;
   // GBK_TO_UNICODE[19265] := 16#7C55;
   // GBK_TO_UNICODE[19266] := 16#BB52;
   // GBK_TO_UNICODE[19267] := 16#7C56;
   // GBK_TO_UNICODE[19268] := 16#BB53;
   // GBK_TO_UNICODE[19269] := 16#7C57;
   // GBK_TO_UNICODE[19270] := 16#BB54;
   // GBK_TO_UNICODE[19271] := 16#7C58;
   // GBK_TO_UNICODE[19272] := 16#BB55;
   // GBK_TO_UNICODE[19273] := 16#7C59;
   // GBK_TO_UNICODE[19274] := 16#BB56;
   // GBK_TO_UNICODE[19275] := 16#7C5A;
   // GBK_TO_UNICODE[19276] := 16#BB57;
   // GBK_TO_UNICODE[19277] := 16#7C5B;
   // GBK_TO_UNICODE[19278] := 16#BB58;
   // GBK_TO_UNICODE[19279] := 16#7C5C;
   // GBK_TO_UNICODE[19280] := 16#BB59;
   // GBK_TO_UNICODE[19281] := 16#7C5D;
   // GBK_TO_UNICODE[19282] := 16#BB5A;
   // GBK_TO_UNICODE[19283] := 16#7C5E;
   // GBK_TO_UNICODE[19284] := 16#BB5B;
   // GBK_TO_UNICODE[19285] := 16#7C5F;
   // GBK_TO_UNICODE[19286] := 16#BB5C;
   // GBK_TO_UNICODE[19287] := 16#7C60;
   // GBK_TO_UNICODE[19288] := 16#BB5D;
   // GBK_TO_UNICODE[19289] := 16#7C61;
   // GBK_TO_UNICODE[19290] := 16#BB5E;
   // GBK_TO_UNICODE[19291] := 16#7C62;
   // GBK_TO_UNICODE[19292] := 16#BB5F;
   // GBK_TO_UNICODE[19293] := 16#7C63;
   // GBK_TO_UNICODE[19294] := 16#BB60;
   // GBK_TO_UNICODE[19295] := 16#7C64;
   // GBK_TO_UNICODE[19296] := 16#BB61;
   // GBK_TO_UNICODE[19297] := 16#7C65;
   // GBK_TO_UNICODE[19298] := 16#BB62;
   // GBK_TO_UNICODE[19299] := 16#7C66;
   // GBK_TO_UNICODE[19300] := 16#BB63;
   // GBK_TO_UNICODE[19301] := 16#7C67;
   // GBK_TO_UNICODE[19302] := 16#BB64;
   // GBK_TO_UNICODE[19303] := 16#7C68;
   // GBK_TO_UNICODE[19304] := 16#BB65;
   // GBK_TO_UNICODE[19305] := 16#7C69;
   // GBK_TO_UNICODE[19306] := 16#BB66;
   // GBK_TO_UNICODE[19307] := 16#7C6A;
   // GBK_TO_UNICODE[19308] := 16#BB67;
   // GBK_TO_UNICODE[19309] := 16#7C6B;
   // GBK_TO_UNICODE[19310] := 16#BB68;
   // GBK_TO_UNICODE[19311] := 16#7C6C;
   // GBK_TO_UNICODE[19312] := 16#BB69;
   // GBK_TO_UNICODE[19313] := 16#7C6D;
   // GBK_TO_UNICODE[19314] := 16#BB6A;
   // GBK_TO_UNICODE[19315] := 16#7C6E;
   // GBK_TO_UNICODE[19316] := 16#BB6B;
   // GBK_TO_UNICODE[19317] := 16#7C6F;
   // GBK_TO_UNICODE[19318] := 16#BB6C;
   // GBK_TO_UNICODE[19319] := 16#7C70;
   // GBK_TO_UNICODE[19320] := 16#BB6D;
   // GBK_TO_UNICODE[19321] := 16#7C71;
   // GBK_TO_UNICODE[19322] := 16#BB6E;
   // GBK_TO_UNICODE[19323] := 16#7C72;
   // GBK_TO_UNICODE[19324] := 16#BB6F;
   // GBK_TO_UNICODE[19325] := 16#7C75;
   // GBK_TO_UNICODE[19326] := 16#BB70;
   // GBK_TO_UNICODE[19327] := 16#7C76;
   // GBK_TO_UNICODE[19328] := 16#BB71;
   // GBK_TO_UNICODE[19329] := 16#7C77;
   // GBK_TO_UNICODE[19330] := 16#BB72;
   // GBK_TO_UNICODE[19331] := 16#7C78;
   // GBK_TO_UNICODE[19332] := 16#BB73;
   // GBK_TO_UNICODE[19333] := 16#7C79;
   // GBK_TO_UNICODE[19334] := 16#BB74;
   // GBK_TO_UNICODE[19335] := 16#7C7A;
   // GBK_TO_UNICODE[19336] := 16#BB75;
   // GBK_TO_UNICODE[19337] := 16#7C7E;
   // GBK_TO_UNICODE[19338] := 16#BB76;
   // GBK_TO_UNICODE[19339] := 16#7C7F;
   // GBK_TO_UNICODE[19340] := 16#BB77;
   // GBK_TO_UNICODE[19341] := 16#7C80;
   // GBK_TO_UNICODE[19342] := 16#BB78;
   // GBK_TO_UNICODE[19343] := 16#7C81;
   // GBK_TO_UNICODE[19344] := 16#BB79;
   // GBK_TO_UNICODE[19345] := 16#7C82;
   // GBK_TO_UNICODE[19346] := 16#BB7A;
   // GBK_TO_UNICODE[19347] := 16#7C83;
   // GBK_TO_UNICODE[19348] := 16#BB7B;
   // GBK_TO_UNICODE[19349] := 16#7C84;
   // GBK_TO_UNICODE[19350] := 16#BB7C;
   // GBK_TO_UNICODE[19351] := 16#7C85;
   // GBK_TO_UNICODE[19352] := 16#BB7D;
   // GBK_TO_UNICODE[19353] := 16#7C86;
   // GBK_TO_UNICODE[19354] := 16#BB7E;
   // GBK_TO_UNICODE[19355] := 16#7C87;
   // GBK_TO_UNICODE[19356] := 16#BB80;
   // GBK_TO_UNICODE[19357] := 16#7C88;
   // GBK_TO_UNICODE[19358] := 16#BB81;
   // GBK_TO_UNICODE[19359] := 16#7C8A;
   // GBK_TO_UNICODE[19360] := 16#BB82;
   // GBK_TO_UNICODE[19361] := 16#7C8B;
   // GBK_TO_UNICODE[19362] := 16#BB83;
   // GBK_TO_UNICODE[19363] := 16#7C8C;
   // GBK_TO_UNICODE[19364] := 16#BB84;
   // GBK_TO_UNICODE[19365] := 16#7C8D;
   // GBK_TO_UNICODE[19366] := 16#BB85;
   // GBK_TO_UNICODE[19367] := 16#7C8E;
   // GBK_TO_UNICODE[19368] := 16#BB86;
   // GBK_TO_UNICODE[19369] := 16#7C8F;
   // GBK_TO_UNICODE[19370] := 16#BB87;
   // GBK_TO_UNICODE[19371] := 16#7C90;
   // GBK_TO_UNICODE[19372] := 16#BB88;
   // GBK_TO_UNICODE[19373] := 16#7C93;
   // GBK_TO_UNICODE[19374] := 16#BB89;
   // GBK_TO_UNICODE[19375] := 16#7C94;
   // GBK_TO_UNICODE[19376] := 16#BB8A;
   // GBK_TO_UNICODE[19377] := 16#7C96;
   // GBK_TO_UNICODE[19378] := 16#BB8B;
   // GBK_TO_UNICODE[19379] := 16#7C99;
   // GBK_TO_UNICODE[19380] := 16#BB8C;
   // GBK_TO_UNICODE[19381] := 16#7C9A;
   // GBK_TO_UNICODE[19382] := 16#BB8D;
   // GBK_TO_UNICODE[19383] := 16#7C9B;
   // GBK_TO_UNICODE[19384] := 16#BB8E;
   // GBK_TO_UNICODE[19385] := 16#7CA0;
   // GBK_TO_UNICODE[19386] := 16#BB8F;
   // GBK_TO_UNICODE[19387] := 16#7CA1;
   // GBK_TO_UNICODE[19388] := 16#BB90;
   // GBK_TO_UNICODE[19389] := 16#7CA3;
   // GBK_TO_UNICODE[19390] := 16#BB91;
   // GBK_TO_UNICODE[19391] := 16#7CA6;
   // GBK_TO_UNICODE[19392] := 16#BB92;
   // GBK_TO_UNICODE[19393] := 16#7CA7;
   // GBK_TO_UNICODE[19394] := 16#BB93;
   // GBK_TO_UNICODE[19395] := 16#7CA8;
   // GBK_TO_UNICODE[19396] := 16#BB94;
   // GBK_TO_UNICODE[19397] := 16#7CA9;
   // GBK_TO_UNICODE[19398] := 16#BB95;
   // GBK_TO_UNICODE[19399] := 16#7CAB;
   // GBK_TO_UNICODE[19400] := 16#BB96;
   // GBK_TO_UNICODE[19401] := 16#7CAC;
   // GBK_TO_UNICODE[19402] := 16#BB97;
   // GBK_TO_UNICODE[19403] := 16#7CAD;
   // GBK_TO_UNICODE[19404] := 16#BB98;
   // GBK_TO_UNICODE[19405] := 16#7CAF;
   // GBK_TO_UNICODE[19406] := 16#BB99;
   // GBK_TO_UNICODE[19407] := 16#7CB0;
   // GBK_TO_UNICODE[19408] := 16#BB9A;
   // GBK_TO_UNICODE[19409] := 16#7CB4;
   // GBK_TO_UNICODE[19410] := 16#BB9B;
   // GBK_TO_UNICODE[19411] := 16#7CB5;
   // GBK_TO_UNICODE[19412] := 16#BB9C;
   // GBK_TO_UNICODE[19413] := 16#7CB6;
   // GBK_TO_UNICODE[19414] := 16#BB9D;
   // GBK_TO_UNICODE[19415] := 16#7CB7;
   // GBK_TO_UNICODE[19416] := 16#BB9E;
   // GBK_TO_UNICODE[19417] := 16#7CB8;
   // GBK_TO_UNICODE[19418] := 16#BB9F;
   // GBK_TO_UNICODE[19419] := 16#7CBA;
   // GBK_TO_UNICODE[19420] := 16#BBA0;
   // GBK_TO_UNICODE[19421] := 16#7CBB;
   // GBK_TO_UNICODE[19422] := 16#BBA1;
   // GBK_TO_UNICODE[19423] := 16#5F27;
   // GBK_TO_UNICODE[19424] := 16#BBA2;
   // GBK_TO_UNICODE[19425] := 16#864E;
   // GBK_TO_UNICODE[19426] := 16#BBA3;
   // GBK_TO_UNICODE[19427] := 16#552C;
   // GBK_TO_UNICODE[19428] := 16#BBA4;
   // GBK_TO_UNICODE[19429] := 16#62A4;
   // GBK_TO_UNICODE[19430] := 16#BBA5;
   // GBK_TO_UNICODE[19431] := 16#4E92;
   // GBK_TO_UNICODE[19432] := 16#BBA6;
   // GBK_TO_UNICODE[19433] := 16#6CAA;
   // GBK_TO_UNICODE[19434] := 16#BBA7;
   // GBK_TO_UNICODE[19435] := 16#6237;
   // GBK_TO_UNICODE[19436] := 16#BBA8;
   // GBK_TO_UNICODE[19437] := 16#82B1;
   // GBK_TO_UNICODE[19438] := 16#BBA9;
   // GBK_TO_UNICODE[19439] := 16#54D7;
   // GBK_TO_UNICODE[19440] := 16#BBAA;
   // GBK_TO_UNICODE[19441] := 16#534E;
   // GBK_TO_UNICODE[19442] := 16#BBAB;
   // GBK_TO_UNICODE[19443] := 16#733E;
   // GBK_TO_UNICODE[19444] := 16#BBAC;
   // GBK_TO_UNICODE[19445] := 16#6ED1;
   // GBK_TO_UNICODE[19446] := 16#BBAD;
   // GBK_TO_UNICODE[19447] := 16#753B;
   // GBK_TO_UNICODE[19448] := 16#BBAE;
   // GBK_TO_UNICODE[19449] := 16#5212;
   // GBK_TO_UNICODE[19450] := 16#BBAF;
   // GBK_TO_UNICODE[19451] := 16#5316;
   // GBK_TO_UNICODE[19452] := 16#BBB0;
   // GBK_TO_UNICODE[19453] := 16#8BDD;
   // GBK_TO_UNICODE[19454] := 16#BBB1;
   // GBK_TO_UNICODE[19455] := 16#69D0;
   // GBK_TO_UNICODE[19456] := 16#BBB2;
   // GBK_TO_UNICODE[19457] := 16#5F8A;
   // GBK_TO_UNICODE[19458] := 16#BBB3;
   // GBK_TO_UNICODE[19459] := 16#6000;
   // GBK_TO_UNICODE[19460] := 16#BBB4;
   // GBK_TO_UNICODE[19461] := 16#6DEE;
   // GBK_TO_UNICODE[19462] := 16#BBB5;
   // GBK_TO_UNICODE[19463] := 16#574F;
   // GBK_TO_UNICODE[19464] := 16#BBB6;
   // GBK_TO_UNICODE[19465] := 16#6B22;
   // GBK_TO_UNICODE[19466] := 16#BBB7;
   // GBK_TO_UNICODE[19467] := 16#73AF;
   // GBK_TO_UNICODE[19468] := 16#BBB8;
   // GBK_TO_UNICODE[19469] := 16#6853;
   // GBK_TO_UNICODE[19470] := 16#BBB9;
   // GBK_TO_UNICODE[19471] := 16#8FD8;
   // GBK_TO_UNICODE[19472] := 16#BBBA;
   // GBK_TO_UNICODE[19473] := 16#7F13;
   // GBK_TO_UNICODE[19474] := 16#BBBB;
   // GBK_TO_UNICODE[19475] := 16#6362;
   // GBK_TO_UNICODE[19476] := 16#BBBC;
   // GBK_TO_UNICODE[19477] := 16#60A3;
   // GBK_TO_UNICODE[19478] := 16#BBBD;
   // GBK_TO_UNICODE[19479] := 16#5524;
   // GBK_TO_UNICODE[19480] := 16#BBBE;
   // GBK_TO_UNICODE[19481] := 16#75EA;
   // GBK_TO_UNICODE[19482] := 16#BBBF;
   // GBK_TO_UNICODE[19483] := 16#8C62;
   // GBK_TO_UNICODE[19484] := 16#BBC0;
   // GBK_TO_UNICODE[19485] := 16#7115;
   // GBK_TO_UNICODE[19486] := 16#BBC1;
   // GBK_TO_UNICODE[19487] := 16#6DA3;
   // GBK_TO_UNICODE[19488] := 16#BBC2;
   // GBK_TO_UNICODE[19489] := 16#5BA6;
   // GBK_TO_UNICODE[19490] := 16#BBC3;
   // GBK_TO_UNICODE[19491] := 16#5E7B;
   // GBK_TO_UNICODE[19492] := 16#BBC4;
   // GBK_TO_UNICODE[19493] := 16#8352;
   // GBK_TO_UNICODE[19494] := 16#BBC5;
   // GBK_TO_UNICODE[19495] := 16#614C;
   // GBK_TO_UNICODE[19496] := 16#BBC6;
   // GBK_TO_UNICODE[19497] := 16#9EC4;
   // GBK_TO_UNICODE[19498] := 16#BBC7;
   // GBK_TO_UNICODE[19499] := 16#78FA;
   // GBK_TO_UNICODE[19500] := 16#BBC8;
   // GBK_TO_UNICODE[19501] := 16#8757;
   // GBK_TO_UNICODE[19502] := 16#BBC9;
   // GBK_TO_UNICODE[19503] := 16#7C27;
   // GBK_TO_UNICODE[19504] := 16#BBCA;
   // GBK_TO_UNICODE[19505] := 16#7687;
   // GBK_TO_UNICODE[19506] := 16#BBCB;
   // GBK_TO_UNICODE[19507] := 16#51F0;
   // GBK_TO_UNICODE[19508] := 16#BBCC;
   // GBK_TO_UNICODE[19509] := 16#60F6;
   // GBK_TO_UNICODE[19510] := 16#BBCD;
   // GBK_TO_UNICODE[19511] := 16#714C;
   // GBK_TO_UNICODE[19512] := 16#BBCE;
   // GBK_TO_UNICODE[19513] := 16#6643;
   // GBK_TO_UNICODE[19514] := 16#BBCF;
   // GBK_TO_UNICODE[19515] := 16#5E4C;
   // GBK_TO_UNICODE[19516] := 16#BBD0;
   // GBK_TO_UNICODE[19517] := 16#604D;
   // GBK_TO_UNICODE[19518] := 16#BBD1;
   // GBK_TO_UNICODE[19519] := 16#8C0E;
   // GBK_TO_UNICODE[19520] := 16#BBD2;
   // GBK_TO_UNICODE[19521] := 16#7070;
   // GBK_TO_UNICODE[19522] := 16#BBD3;
   // GBK_TO_UNICODE[19523] := 16#6325;
   // GBK_TO_UNICODE[19524] := 16#BBD4;
   // GBK_TO_UNICODE[19525] := 16#8F89;
   // GBK_TO_UNICODE[19526] := 16#BBD5;
   // GBK_TO_UNICODE[19527] := 16#5FBD;
   // GBK_TO_UNICODE[19528] := 16#BBD6;
   // GBK_TO_UNICODE[19529] := 16#6062;
   // GBK_TO_UNICODE[19530] := 16#BBD7;
   // GBK_TO_UNICODE[19531] := 16#86D4;
   // GBK_TO_UNICODE[19532] := 16#BBD8;
   // GBK_TO_UNICODE[19533] := 16#56DE;
   // GBK_TO_UNICODE[19534] := 16#BBD9;
   // GBK_TO_UNICODE[19535] := 16#6BC1;
   // GBK_TO_UNICODE[19536] := 16#BBDA;
   // GBK_TO_UNICODE[19537] := 16#6094;
   // GBK_TO_UNICODE[19538] := 16#BBDB;
   // GBK_TO_UNICODE[19539] := 16#6167;
   // GBK_TO_UNICODE[19540] := 16#BBDC;
   // GBK_TO_UNICODE[19541] := 16#5349;
   // GBK_TO_UNICODE[19542] := 16#BBDD;
   // GBK_TO_UNICODE[19543] := 16#60E0;
   // GBK_TO_UNICODE[19544] := 16#BBDE;
   // GBK_TO_UNICODE[19545] := 16#6666;
   // GBK_TO_UNICODE[19546] := 16#BBDF;
   // GBK_TO_UNICODE[19547] := 16#8D3F;
   // GBK_TO_UNICODE[19548] := 16#BBE0;
   // GBK_TO_UNICODE[19549] := 16#79FD;
   // GBK_TO_UNICODE[19550] := 16#BBE1;
   // GBK_TO_UNICODE[19551] := 16#4F1A;
   // GBK_TO_UNICODE[19552] := 16#BBE2;
   // GBK_TO_UNICODE[19553] := 16#70E9;
   // GBK_TO_UNICODE[19554] := 16#BBE3;
   // GBK_TO_UNICODE[19555] := 16#6C47;
   // GBK_TO_UNICODE[19556] := 16#BBE4;
   // GBK_TO_UNICODE[19557] := 16#8BB3;
   // GBK_TO_UNICODE[19558] := 16#BBE5;
   // GBK_TO_UNICODE[19559] := 16#8BF2;
   // GBK_TO_UNICODE[19560] := 16#BBE6;
   // GBK_TO_UNICODE[19561] := 16#7ED8;
   // GBK_TO_UNICODE[19562] := 16#BBE7;
   // GBK_TO_UNICODE[19563] := 16#8364;
   // GBK_TO_UNICODE[19564] := 16#BBE8;
   // GBK_TO_UNICODE[19565] := 16#660F;
   // GBK_TO_UNICODE[19566] := 16#BBE9;
   // GBK_TO_UNICODE[19567] := 16#5A5A;
